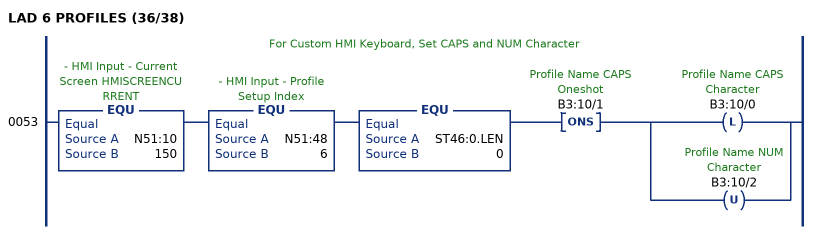
% Rung: 53 %
% For Custom HMI Keyboard, Set CAPS and NUM Character %
SOR EQU N51:10 150 EQU N51:48 6 EQU ST46:0.LEN 0 ONS B3:10/1 BST OTL B3:10/0 NXB OTU B3:10/2 BND EOR
%   N51:10  HMISCREENCURRENT  "- HMI Input - Current Screen" %
%   N51:48  "- HMI Input - Profile Setup Index" %
%   B3:10/1  "Profile Name CAPS Oneshot" %
%   B3:10/0  "Profile Name CAPS Character" %
%   B3:10/2  "Profile Name NUM Character" %

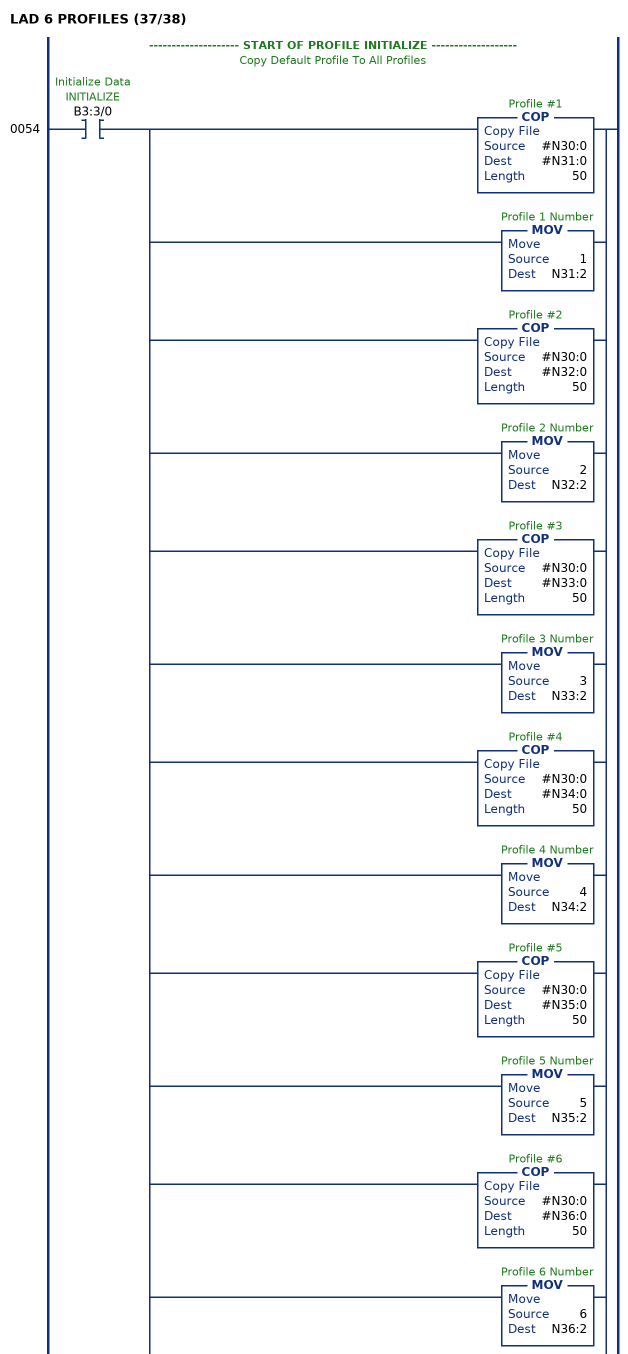

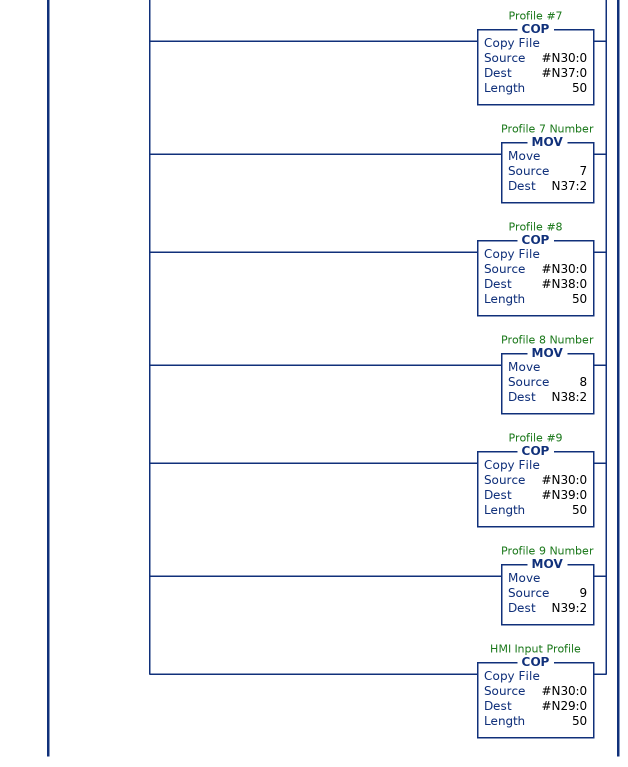
% Rung: 54 %
% TITLE: -------------------- START OF PROFILE INITIALIZE ------------------- %
% Copy Default Profile To All Profiles %
SOR XIC B3:3/0 BST COP #N30:0 #N31:0 50 NXB MOV 1 N31:2 NXB COP #N30:0 #N32:0 50 NXB MOV 2 N32:2 NXB COP #N30:0 #N33:0 50 NXB MOV 3 N33:2 NXB COP #N30:0 #N34:0 50 NXB MOV 4 N34:2 NXB COP #N30:0 #N35:0 50 NXB MOV 5 N35:2 NXB COP #N30:0 #N36:0 50 NXB MOV 6 N36:2 NXB COP #N30:0 #N37:0 50 NXB MOV 7 N37:2 NXB COP #N30:0 #N38:0 50 NXB MOV 8 N38:2 NXB COP #N30:0 #N39:0 50 NXB MOV 9 N39:2 NXB COP #N30:0 #N29:0 50 BND EOR
%   B3:3/0  INITIALIZE  "Initialize Data" %
%   N30:0  "Enable bits" %
%   N31:0  "Profile #1" %
%   N31:2  "Profile 1 Number" %
%   N32:0  "Profile #2" %
%   N32:2  "Profile 2 Number" %
%   N33:0  "Profile #3" %
%   N33:2  "Profile 3 Number" %
%   N34:0  "Profile #4" %
%   N34:2  "Profile 4 Number" %
%   N35:0  "Profile #5" %
%   N35:2  "Profile 5 Number" %
%   N36:0  "Profile #6" %
%   N36:2  "Profile 6 Number" %
%   N37:0  "Profile #7" %
%   N37:2  "Profile 7 Number" %
%   N38:0  "Profile #8" %
%   N38:2  "Profile 8 Number" %
%   N39:0  "Profile #9" %
%   N39:2  "Profile 9 Number" %
%   N29:0  "HMI Input Profile" %

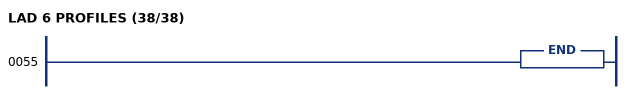
% Rung: 55 %
SOR END EOR

LADDER 7 "OPTIONS"
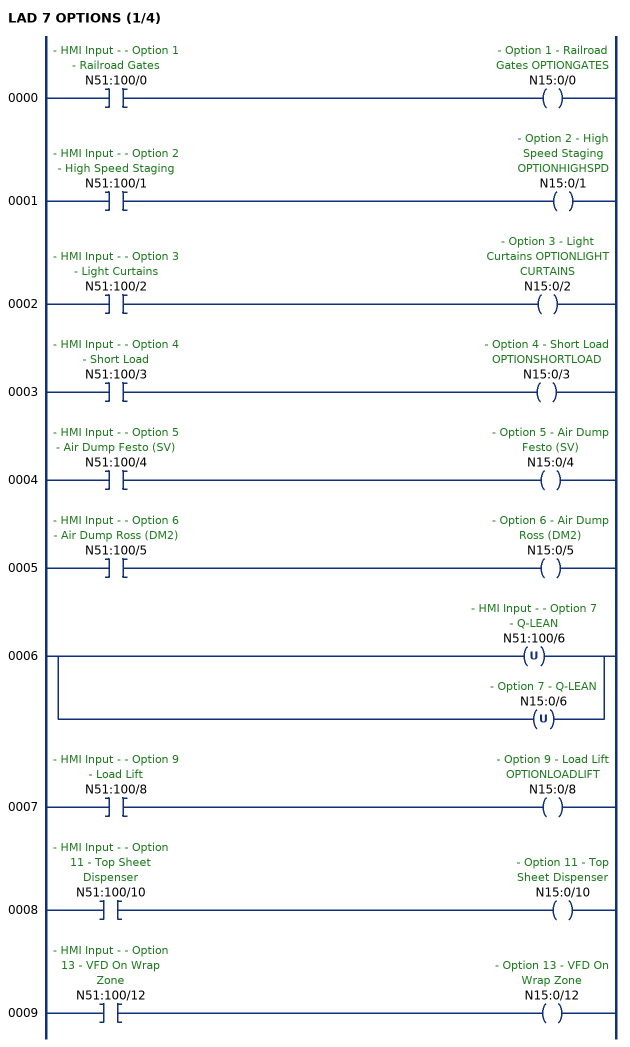
% Rung: 0 %
SOR XIC N51:100/0 OTE N15:0/0 EOR
%   N51:100/0  "- HMI Input - - Option 1 - Railroad Gates" %
%   N15:0/0  OPTIONGATES  "- Option 1 - Railroad Gates" %
% Rung: 1 %
SOR XIC N51:100/1 OTE N15:0/1 EOR
%   N51:100/1  "- HMI Input - - Option 2 - High Speed Staging" %
%   N15:0/1  OPTIONHIGHSPD  "- Option 2 - High Speed Staging" %
% Rung: 2 %
SOR XIC N51:100/2 OTE N15:0/2 EOR
%   N51:100/2  "- HMI Input - - Option 3 - Light Curtains" %
%   N15:0/2  OPTIONLIGHTCURTAINS  "- Option 3 - Light Curtains" %
% Rung: 3 %
SOR XIC N51:100/3 OTE N15:0/3 EOR
%   N51:100/3  "- HMI Input - - Option 4 - Short Load" %
%   N15:0/3  OPTIONSHORTLOAD  "- Option 4 - Short Load" %
% Rung: 4 %
SOR XIC N51:100/4 OTE N15:0/4 EOR
%   N51:100/4  "- HMI Input - - Option 5 - Air Dump Festo (SV)" %
%   N15:0/4  "- Option 5 - Air Dump Festo (SV)" %
% Rung: 5 %
SOR XIC N51:100/5 OTE N15:0/5 EOR
%   N51:100/5  "- HMI Input - - Option 6 - Air Dump Ross (DM2)" %
%   N15:0/5  "- Option 6 - Air Dump Ross (DM2)" %
% Rung: 6 %
SOR BST OTU N51:100/6 NXB OTU N15:0/6 BND EOR
%   N51:100/6  "- HMI Input - - Option 7 - Q-LEAN" %
%   N15:0/6  "- Option 7 - Q-LEAN" %
% Rung: 7 %
SOR XIC N51:100/8 OTE N15:0/8 EOR
%   N51:100/8  "- HMI Input - - Option 9 - Load Lift" %
%   N15:0/8  OPTIONLOADLIFT  "- Option 9 - Load Lift" %
% Rung: 8 %
SOR XIC N51:100/10 OTE N15:0/10 EOR
%   N51:100/10  "- HMI Input - - Option 11 - Top Sheet Dispenser" %
%   N15:0/10  "- Option 11 - Top Sheet Dispenser" %
% Rung: 9 %
SOR XIC N51:100/12 OTE N15:0/12 EOR
%   N51:100/12  "- HMI Input - - Option 13 - VFD On Wrap Zone" %
%   N15:0/12  "- Option 13 - VFD On Wrap Zone" %

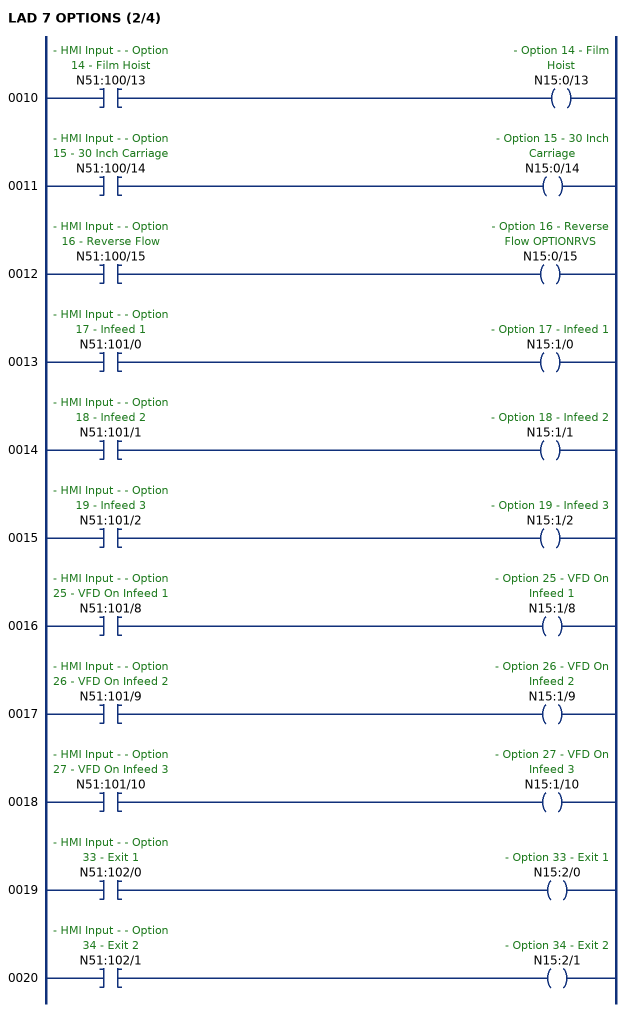
% Rung: 10 %
SOR XIC N51:100/13 OTE N15:0/13 EOR
%   N51:100/13  "- HMI Input - - Option 14 - Film Hoist" %
%   N15:0/13  "- Option 14 - Film Hoist" %
% Rung: 11 %
SOR XIC N51:100/14 OTE N15:0/14 EOR
%   N51:100/14  "- HMI Input - - Option 15 - 30 Inch Carriage" %
%   N15:0/14  "- Option 15 - 30 Inch Carriage" %
% Rung: 12 %
SOR XIC N51:100/15 OTE N15:0/15 EOR
%   N51:100/15  "- HMI Input - - Option 16 - Reverse Flow" %
%   N15:0/15  OPTIONRVS  "- Option 16 - Reverse Flow" %
% Rung: 13 %
SOR XIC N51:101/0 OTE N15:1/0 EOR
%   N51:101/0  "- HMI Input - - Option 17 - Infeed 1" %
%   N15:1/0  "- Option 17 - Infeed 1" %
% Rung: 14 %
SOR XIC N51:101/1 OTE N15:1/1 EOR
%   N51:101/1  "- HMI Input - - Option 18 - Infeed 2" %
%   N15:1/1  "- Option 18 - Infeed 2" %
% Rung: 15 %
SOR XIC N51:101/2 OTE N15:1/2 EOR
%   N51:101/2  "- HMI Input - - Option 19 - Infeed 3" %
%   N15:1/2  "- Option 19 - Infeed 3" %
% Rung: 16 %
SOR XIC N51:101/8 OTE N15:1/8 EOR
%   N51:101/8  "- HMI Input - - Option 25 - VFD On Infeed 1" %
%   N15:1/8  "- Option 25 - VFD On Infeed 1" %
% Rung: 17 %
SOR XIC N51:101/9 OTE N15:1/9 EOR
%   N51:101/9  "- HMI Input - - Option 26 - VFD On Infeed 2" %
%   N15:1/9  "- Option 26 - VFD On Infeed 2" %
% Rung: 18 %
SOR XIC N51:101/10 OTE N15:1/10 EOR
%   N51:101/10  "- HMI Input - - Option 27 - VFD On Infeed 3" %
%   N15:1/10  "- Option 27 - VFD On Infeed 3" %
% Rung: 19 %
SOR XIC N51:102/0 OTE N15:2/0 EOR
%   N51:102/0  "- HMI Input - - Option 33 - Exit 1" %
%   N15:2/0  "- Option 33 - Exit 1" %
% Rung: 20 %
SOR XIC N51:102/1 OTE N15:2/1 EOR
%   N51:102/1  "- HMI Input - - Option 34 - Exit 2" %
%   N15:2/1  "- Option 34 - Exit 2" %

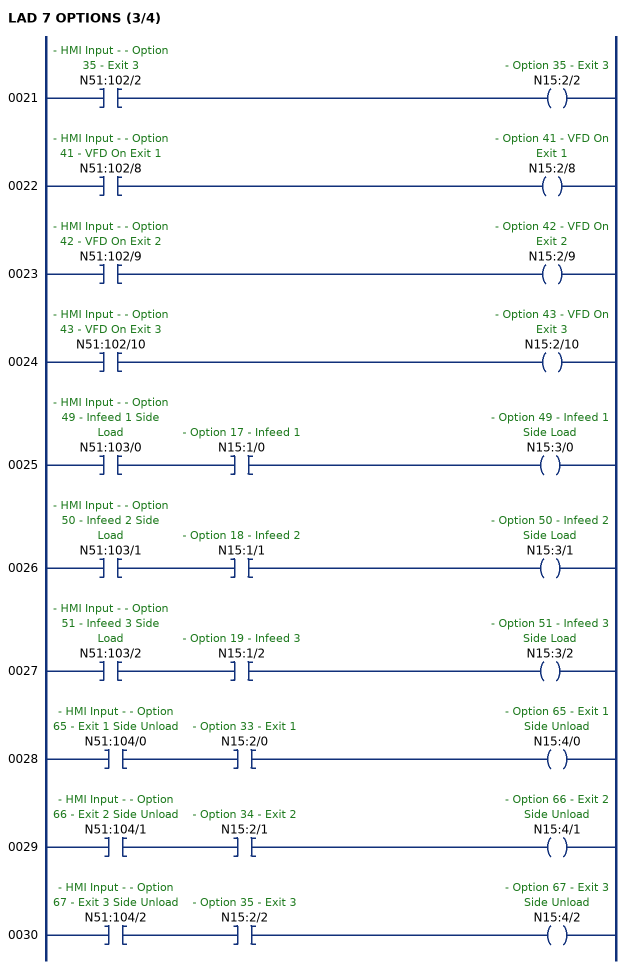
% Rung: 21 %
SOR XIC N51:102/2 OTE N15:2/2 EOR
%   N51:102/2  "- HMI Input - - Option 35 - Exit 3" %
%   N15:2/2  "- Option 35 - Exit 3" %
% Rung: 22 %
SOR XIC N51:102/8 OTE N15:2/8 EOR
%   N51:102/8  "- HMI Input - - Option 41 - VFD On Exit 1" %
%   N15:2/8  "- Option 41 - VFD On Exit 1" %
% Rung: 23 %
SOR XIC N51:102/9 OTE N15:2/9 EOR
%   N51:102/9  "- HMI Input - - Option 42 - VFD On Exit 2" %
%   N15:2/9  "- Option 42 - VFD On Exit 2" %
% Rung: 24 %
SOR XIC N51:102/10 OTE N15:2/10 EOR
%   N51:102/10  "- HMI Input - - Option 43 - VFD On Exit 3" %
%   N15:2/10  "- Option 43 - VFD On Exit 3" %
% Rung: 25 %
SOR XIC N51:103/0 XIC N15:1/0 OTE N15:3/0 EOR
%   N51:103/0  "- HMI Input - - Option 49 - Infeed 1 Side Load" %
%   N15:1/0  "- Option 17 - Infeed 1" %
%   N15:3/0  "- Option 49 - Infeed 1 Side Load" %
% Rung: 26 %
SOR XIC N51:103/1 XIC N15:1/1 OTE N15:3/1 EOR
%   N51:103/1  "- HMI Input - - Option 50 - Infeed 2 Side Load" %
%   N15:1/1  "- Option 18 - Infeed 2" %
%   N15:3/1  "- Option 50 - Infeed 2 Side Load" %
% Rung: 27 %
SOR XIC N51:103/2 XIC N15:1/2 OTE N15:3/2 EOR
%   N51:103/2  "- HMI Input - - Option 51 - Infeed 3 Side Load" %
%   N15:1/2  "- Option 19 - Infeed 3" %
%   N15:3/2  "- Option 51 - Infeed 3 Side Load" %
% Rung: 28 %
SOR XIC N51:104/0 XIC N15:2/0 OTE N15:4/0 EOR
%   N51:104/0  "- HMI Input - - Option 65 - Exit 1 Side Unload" %
%   N15:2/0  "- Option 33 - Exit 1" %
%   N15:4/0  "- Option 65 - Exit 1 Side Unload" %
% Rung: 29 %
SOR XIC N51:104/1 XIC N15:2/1 OTE N15:4/1 EOR
%   N51:104/1  "- HMI Input - - Option 66 - Exit 2 Side Unload" %
%   N15:2/1  "- Option 34 - Exit 2" %
%   N15:4/1  "- Option 66 - Exit 2 Side Unload" %
% Rung: 30 %
SOR XIC N51:104/2 XIC N15:2/2 OTE N15:4/2 EOR
%   N51:104/2  "- HMI Input - - Option 67 - Exit 3 Side Unload" %
%   N15:2/2  "- Option 35 - Exit 3" %
%   N15:4/2  "- Option 67 - Exit 3 Side Unload" %

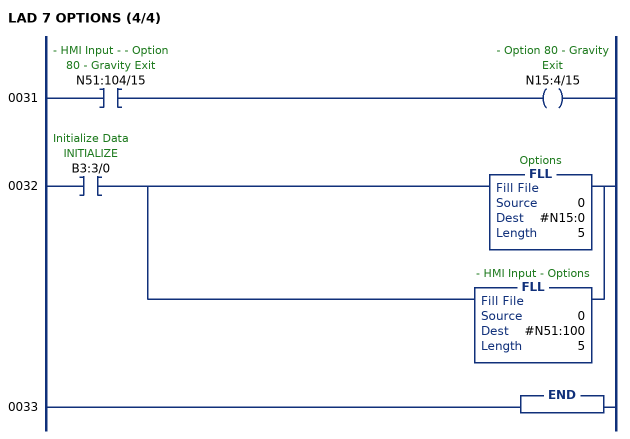
% Rung: 31 %
SOR XIC N51:104/15 OTE N15:4/15 EOR
%   N51:104/15  "- HMI Input - - Option 80 - Gravity Exit" %
%   N15:4/15  "- Option 80 - Gravity Exit" %
% Rung: 32 %
SOR XIC B3:3/0 BST FLL 0 #N15:0 5 NXB FLL 0 #N51:100 5 BND EOR
%   B3:3/0  INITIALIZE  "Initialize Data" %
%   N15:0  "Options" %
%   N51:100  "- HMI Input - Options" %
% Rung: 33 %
SOR END EOR

LADDER 8 "CONSTANTS"
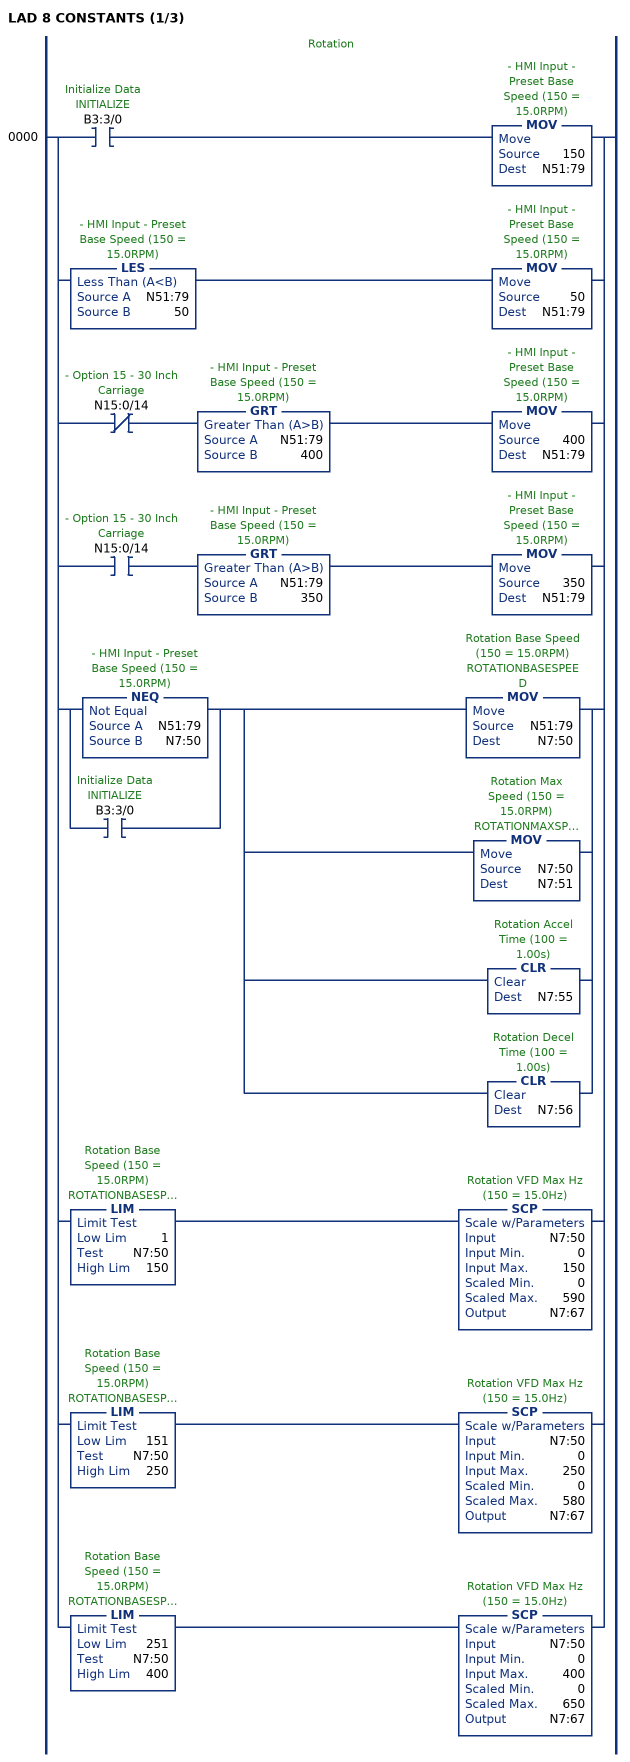
% Rung: 0 %
% Rotation %
SOR BST BST XIC B3:3/0 MOV 150 N51:79 NXB LES N51:79 50 MOV 50 N51:79 NXB XIO N15:0/14 GRT N51:79 400 MOV 400 N51:79 NXB XIC N15:0/14 GRT N51:79 350 MOV 350 N51:79 BND NXB BST NEQ N51:79 N7:50 NXB XIC B3:3/0 BND BST MOV N51:79 N7:50 NXB MOV N7:50 N7:51 NXB CLR N7:55 NXB CLR N7:56 BND NXB BST LIM 1 N7:50 150 SCP N7:50 0 150 0 590 N7:67 NXB LIM 151 N7:50 250 SCP N7:50 0 250 0 580 N7:67 NXB LIM 251 N7:50 400 SCP N7:50 0 400 0 650 N7:67 BND BND EOR
%   B3:3/0  INITIALIZE  "Initialize Data" %
%   N51:79  "- HMI Input - Preset Base Speed (150 = 15.0RPM)" %
%   N15:0/14  "- Option 15 - 30 Inch Carriage" %
%   N7:50  ROTATIONBASESPEED  "Rotation Base Speed (150 = 15.0RPM)" %
%   N7:51  ROTATIONMAXSPEED  "Rotation Max Speed (150 = 15.0RPM)" %
%   N7:55  "Rotation Accel Time (100 = 1.00s)" %
%   N7:56  "Rotation Decel Time (100 = 1.00s)" %
%   N7:67  "Rotation VFD Max Hz (150 = 15.0Hz)" %

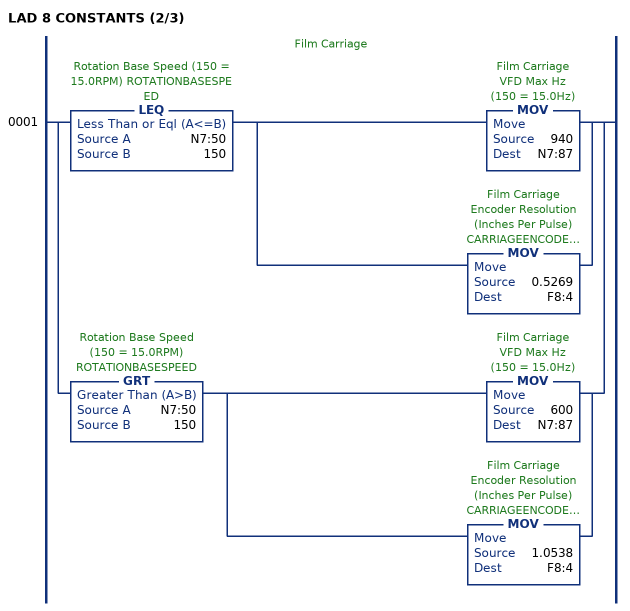
% Rung: 1 %
% Film Carriage %
SOR BST LEQ N7:50 150 BST MOV 940 N7:87 NXB MOV 0.5269 F8:4 BND NXB GRT N7:50 150 BST MOV 600 N7:87 NXB MOV 1.0538 F8:4 BND BND EOR
%   N7:50  ROTATIONBASESPEED  "Rotation Base Speed (150 = 15.0RPM)" %
%   N7:87  "Film Carriage VFD Max Hz (150 = 15.0Hz)" %
%   F8:4  CARRIAGEENCODERRES  "Film Carriage Encoder Resolution (Inches Per Pulse)" %

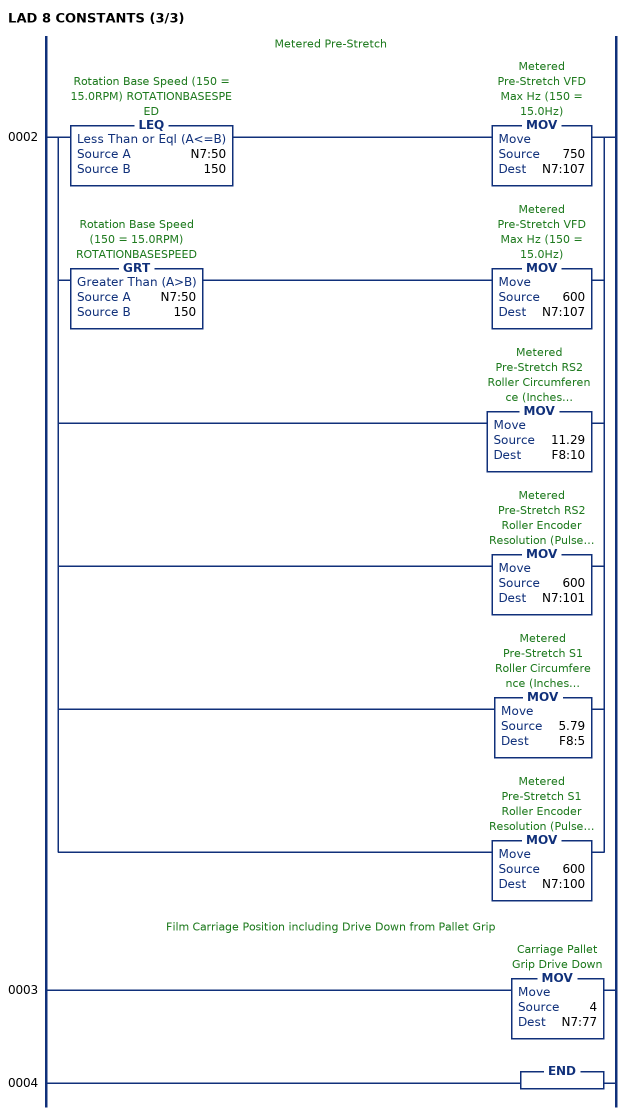
% Rung: 2 %
% Metered Pre-Stretch %
SOR BST BST LEQ N7:50 150 MOV 750 N7:107 NXB GRT N7:50 150 MOV 600 N7:107 BND NXB MOV 11.29 F8:10 NXB MOV 600 N7:101 NXB MOV 5.79 F8:5 NXB MOV 600 N7:100 BND EOR
%   N7:50  ROTATIONBASESPEED  "Rotation Base Speed (150 = 15.0RPM)" %
%   N7:107  "Metered Pre-Stretch VFD Max Hz (150 = 15.0Hz)" %
%   F8:10  MPSRS2CIRC  "Metered Pre-Stretch RS2 Roller Circumference (Inches)" %
%   N7:101  MPSRS2ENCODERRES  "Metered Pre-Stretch RS2 Roller Encoder Resolution (Pulses Per Rev)" %
%   F8:5  MPSS1CIRC  "Metered Pre-Stretch S1 Roller Circumference (Inches)" %
%   N7:100  MPSS1ENCODERRES  "Metered Pre-Stretch S1 Roller Encoder Resolution (Pulses Per Rev)" %
% Rung: 3 %
% Film Carriage Position including Drive Down from Pallet Grip %
SOR MOV 4 N7:77 EOR
%   N7:77  "Carriage Pallet Grip Drive Down" %
% Rung: 4 %
SOR END EOR

LADDER 9 "WRAP CYCLE"
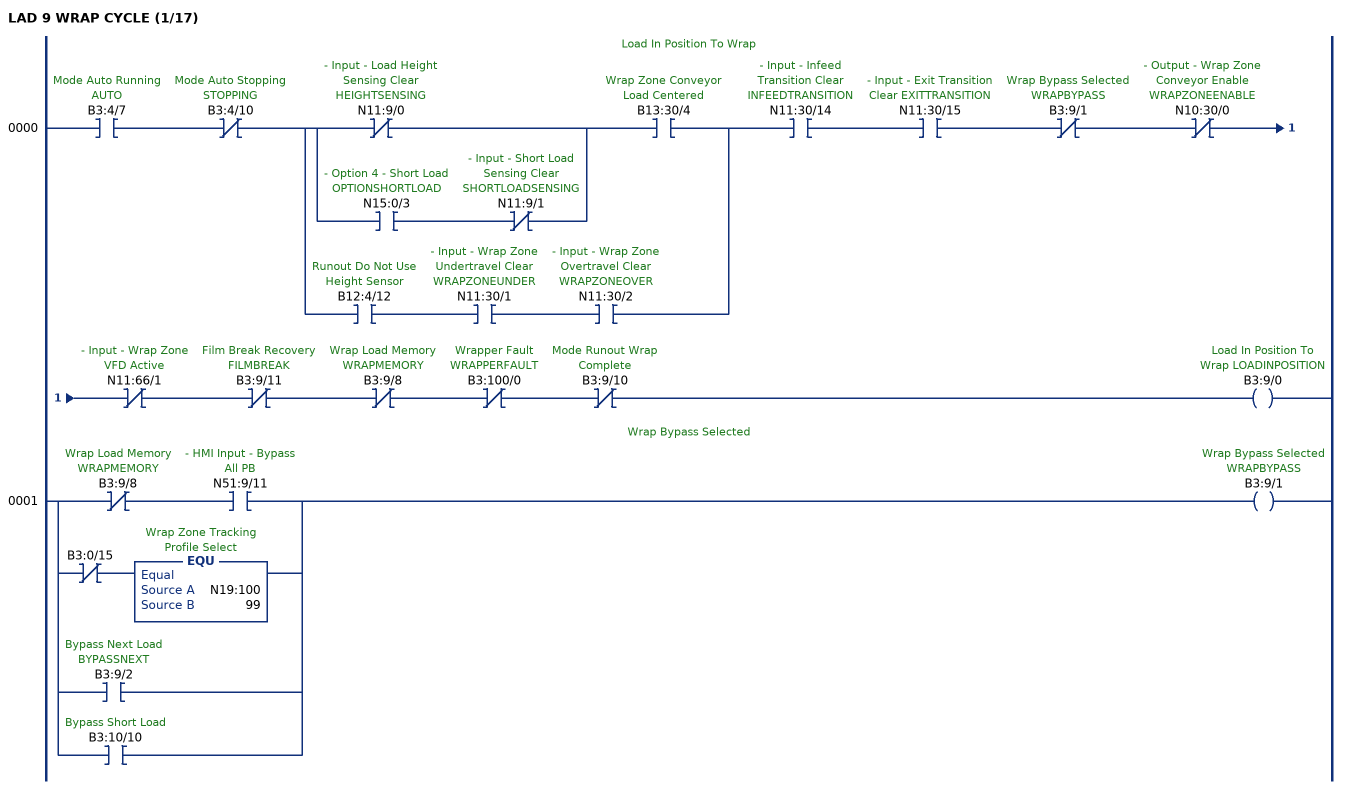
% Rung: 0 %
% Load In Position To Wrap %
SOR XIC B3:4/7 XIO B3:4/10 BST BST XIO N11:9/0 NXB XIC N15:0/3 XIO N11:9/1 BND XIC B13:30/4 NXB XIC B12:4/12 XIC N11:30/1 XIC N11:30/2 BND XIC N11:30/14 XIC N11:30/15 XIO B3:9/1 XIO N10:30/0 XIO N11:66/1 XIO B3:9/11 XIO B3:9/8 XIO B3:100/0 XIO B3:9/10 OTE B3:9/0 EOR
%   B3:4/7  AUTO  "Mode Auto Running" %
%   B3:4/10  STOPPING  "Mode Auto Stopping" %
%   N11:9/0  HEIGHTSENSING  "- Input - Load Height Sensing Clear" %
%   N15:0/3  OPTIONSHORTLOAD  "- Option 4 - Short Load" %
%   N11:9/1  SHORTLOADSENSING  "- Input - Short Load Sensing Clear" %
%   B13:30/4  "Wrap Zone Conveyor Load Centered" %
%   B12:4/12  "Runout Do Not Use Height Sensor" %
%   N11:30/1  WRAPZONEUNDER  "- Input - Wrap Zone Undertravel Clear" %
%   N11:30/2  WRAPZONEOVER  "- Input - Wrap Zone Overtravel Clear" %
%   N11:30/14  INFEEDTRANSITION  "- Input - Infeed Transition Clear" %
%   N11:30/15  EXITTRANSITION  "- Input - Exit Transition Clear" %
%   B3:9/1  WRAPBYPASS  "Wrap Bypass Selected" %
%   N10:30/0  WRAPZONEENABLE  "- Output - Wrap Zone Conveyor Enable" %
%   N11:66/1  "- Input - Wrap Zone VFD Active" %
%   B3:9/11  FILMBREAK  "Film Break Recovery" %
%   B3:9/8  WRAPMEMORY  "Wrap Load Memory" %
%   B3:100/0  WRAPPERFAULT  "Wrapper Fault" %
%   B3:9/10  "Mode Runout Wrap Complete" %
%   B3:9/0  LOADINPOSITION  "Load In Position To Wrap" %
% Rung: 1 %
% Wrap Bypass Selected %
SOR BST XIO B3:9/8 XIC N51:9/11 NXB XIO B3:0/15 EQU N19:100 99 NXB XIC B3:9/2 NXB XIC B3:10/10 BND OTE B3:9/1 EOR
%   B3:9/8  WRAPMEMORY  "Wrap Load Memory" %
%   N51:9/11  "- HMI Input - Bypass All PB" %
%   N19:100  "Wrap Zone Tracking Profile Select" %
%   B3:9/2  BYPASSNEXT  "Bypass Next Load" %
%   B3:10/10  "Bypass Short Load" %
%   B3:9/1  WRAPBYPASS  "Wrap Bypass Selected" %

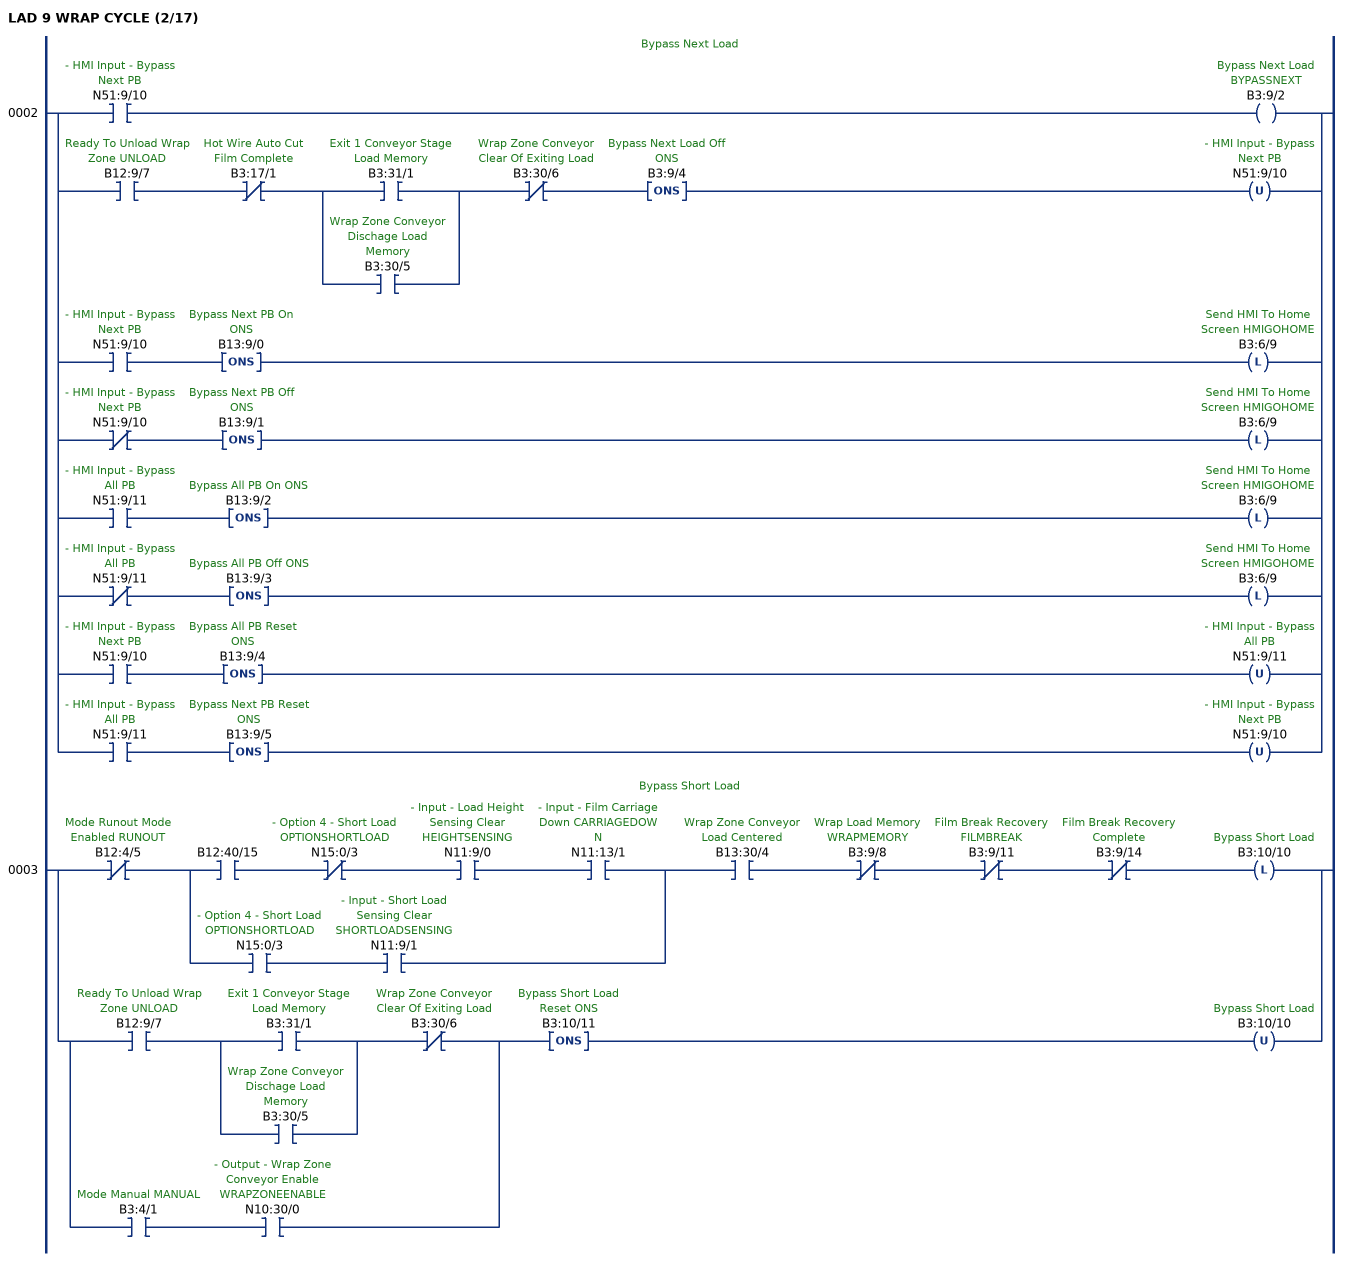
% Rung: 2 %
% Bypass Next Load %
SOR BST XIC N51:9/10 OTE B3:9/2 NXB XIC B12:9/7 XIO B3:17/1 BST XIC B3:31/1 NXB XIC B3:30/5 BND XIO B3:30/6 ONS B3:9/4 OTU N51:9/10 NXB BST XIC N51:9/10 ONS B13:9/0 OTL B3:6/9 NXB XIO N51:9/10 ONS B13:9/1 OTL B3:6/9 NXB XIC N51:9/11 ONS B13:9/2 OTL B3:6/9 NXB XIO N51:9/11 ONS B13:9/3 OTL B3:6/9 BND NXB BST XIC N51:9/10 ONS B13:9/4 OTU N51:9/11 NXB XIC N51:9/11 ONS B13:9/5 OTU N51:9/10 BND BND EOR
%   N51:9/10  "- HMI Input - Bypass Next PB" %
%   B3:9/2  BYPASSNEXT  "Bypass Next Load" %
%   B12:9/7  UNLOAD  "Ready To Unload Wrap Zone" %
%   B3:17/1  "Hot Wire Auto Cut Film Complete" %
%   B3:31/1  "Exit 1 Conveyor Stage Load Memory" %
%   B3:30/5  "Wrap Zone Conveyor Dischage Load Memory" %
%   B3:30/6  "Wrap Zone Conveyor Clear Of Exiting Load" %
%   B3:9/4  "Bypass Next Load Off ONS" %
%   B13:9/0  "Bypass Next PB On ONS" %
%   B3:6/9  HMIGOHOME  "Send HMI To Home Screen" %
%   B13:9/1  "Bypass Next PB Off ONS" %
%   N51:9/11  "- HMI Input - Bypass All PB" %
%   B13:9/2  "Bypass All PB On ONS" %
%   B13:9/3  "Bypass All PB Off ONS" %
%   B13:9/4  "Bypass All PB Reset ONS" %
%   B13:9/5  "Bypass Next PB Reset ONS" %
% Rung: 3 %
% Bypass Short Load %
SOR BST XIO B12:4/5 BST XIC B12:40/15 XIO N15:0/3 XIC N11:9/0 XIC N11:13/1 NXB XIC N15:0/3 XIC N11:9/1 BND XIC B13:30/4 XIO B3:9/8 XIO B3:9/11 XIO B3:9/14 OTL B3:10/10 NXB BST XIC B12:9/7 BST XIC B3:31/1 NXB XIC B3:30/5 BND XIO B3:30/6 NXB XIC B3:4/1 XIC N10:30/0 BND ONS B3:10/11 OTU B3:10/10 BND EOR
%   B12:4/5  RUNOUT  "Mode Runout Mode Enabled" %
%   N15:0/3  OPTIONSHORTLOAD  "- Option 4 - Short Load" %
%   N11:9/0  HEIGHTSENSING  "- Input - Load Height Sensing Clear" %
%   N11:13/1  CARRIAGEDOWN  "- Input - Film Carriage Down" %
%   N11:9/1  SHORTLOADSENSING  "- Input - Short Load Sensing Clear" %
%   B13:30/4  "Wrap Zone Conveyor Load Centered" %
%   B3:9/8  WRAPMEMORY  "Wrap Load Memory" %
%   B3:9/11  FILMBREAK  "Film Break Recovery" %
%   B3:9/14  "Film Break Recovery Complete" %
%   B3:10/10  "Bypass Short Load" %
%   B12:9/7  UNLOAD  "Ready To Unload Wrap Zone" %
%   B3:31/1  "Exit 1 Conveyor Stage Load Memory" %
%   B3:30/5  "Wrap Zone Conveyor Dischage Load Memory" %
%   B3:30/6  "Wrap Zone Conveyor Clear Of Exiting Load" %
%   B3:4/1  MANUAL  "Mode Manual" %
%   N10:30/0  WRAPZONEENABLE  "- Output - Wrap Zone Conveyor Enable" %
%   B3:10/11  "Bypass Short Load Reset ONS" %

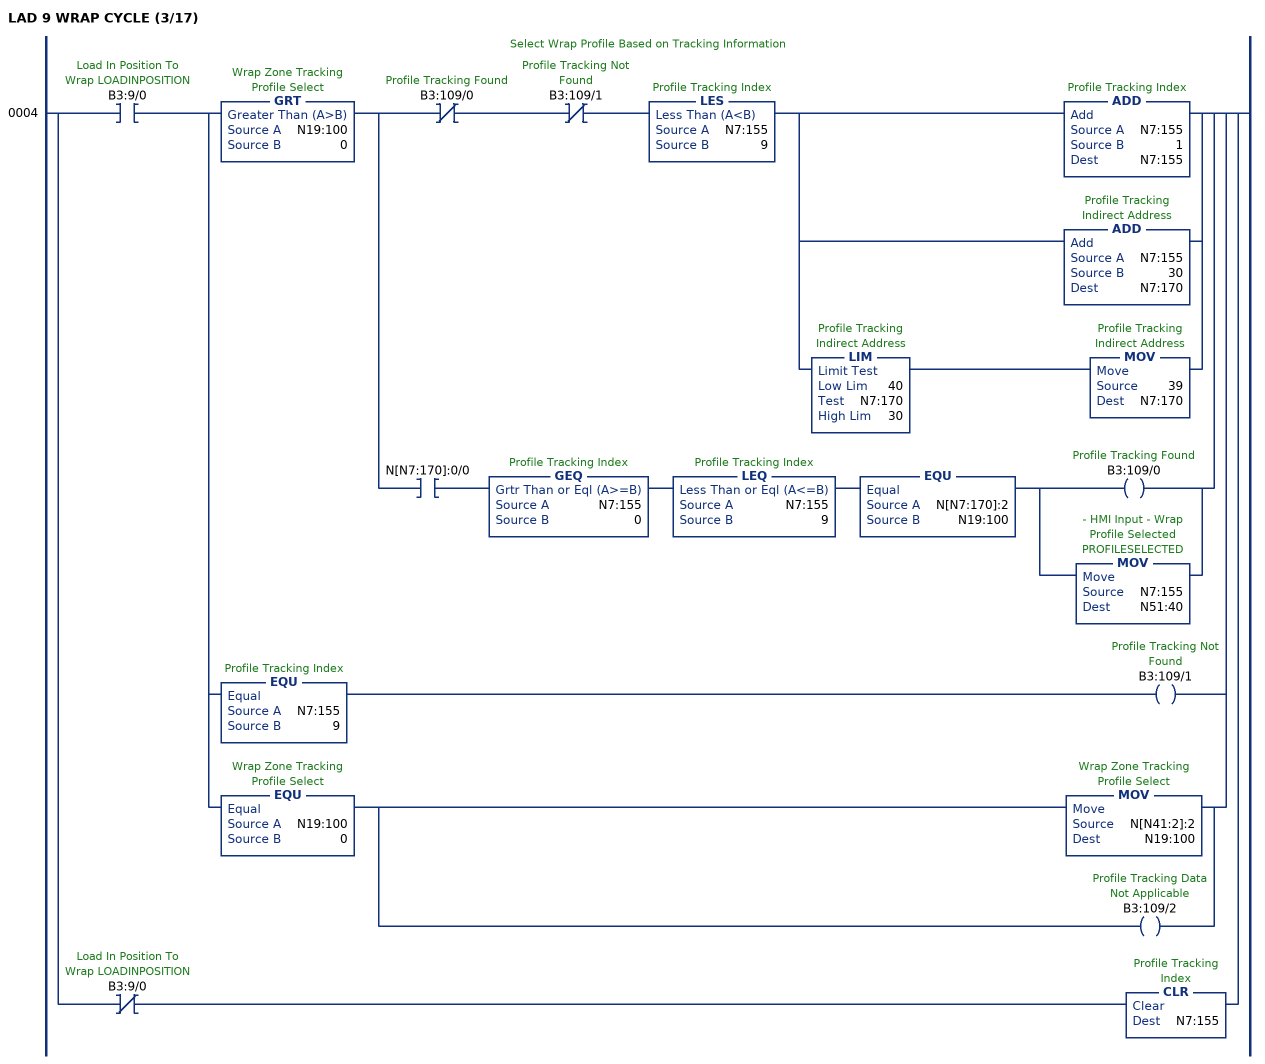
% Rung: 4 %
% Select Wrap Profile Based on Tracking Information %
SOR BST XIC B3:9/0 BST GRT N19:100 0 BST XIO B3:109/0 XIO B3:109/1 LES N7:155 9 BST ADD N7:155 1 N7:155 NXB ADD N7:155 30 N7:170 NXB LIM 40 N7:170 30 MOV 39 N7:170 BND NXB XIC N[N7:170]:0/0 GEQ N7:155 0 LEQ N7:155 9 EQU N[N7:170]:2 N19:100 BST OTE B3:109/0 NXB MOV N7:155 N51:40 BND BND NXB EQU N7:155 9 OTE B3:109/1 NXB EQU N19:100 0 BST MOV N[N41:2]:2 N19:100 NXB OTE B3:109/2 BND BND NXB XIO B3:9/0 CLR N7:155 BND EOR
%   B3:9/0  LOADINPOSITION  "Load In Position To Wrap" %
%   N19:100  "Wrap Zone Tracking Profile Select" %
%   B3:109/0  "Profile Tracking Found" %
%   B3:109/1  "Profile Tracking Not Found" %
%   N7:155  "Profile Tracking Index" %
%   N7:170  "Profile Tracking Indirect Address" %
%   N51:40  PROFILESELECTED  "- HMI Input - Wrap Profile Selected" %
%   N41:2  "Profile Selected Indirect Address" %
%   B3:109/2  "Profile Tracking Data Not Applicable" %

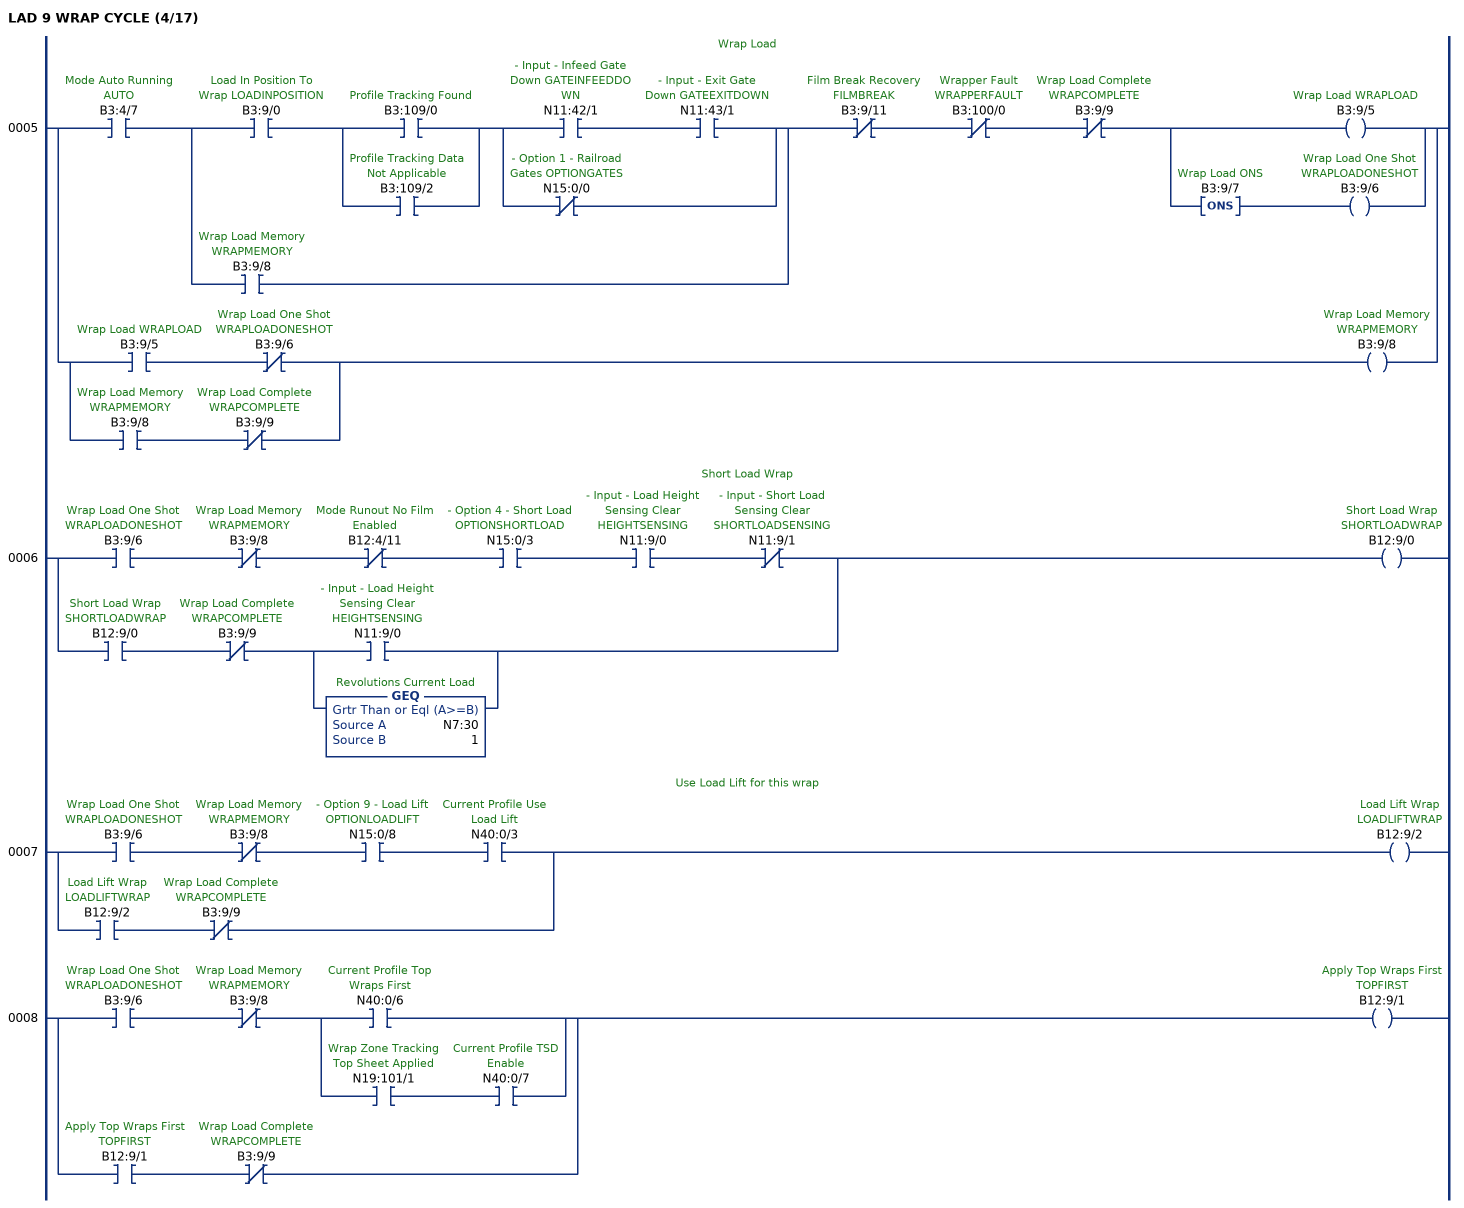
% Rung: 5 %
% Wrap Load %
SOR BST XIC B3:4/7 BST XIC B3:9/0 BST XIC B3:109/0 NXB XIC B3:109/2 BND BST XIC N11:42/1 XIC N11:43/1 NXB XIO N15:0/0 BND NXB XIC B3:9/8 BND XIO B3:9/11 XIO B3:100/0 XIO B3:9/9 BST OTE B3:9/5 NXB ONS B3:9/7 OTE B3:9/6 BND NXB BST XIC B3:9/5 XIO B3:9/6 NXB XIC B3:9/8 XIO B3:9/9 BND OTE B3:9/8 BND EOR
%   B3:4/7  AUTO  "Mode Auto Running" %
%   B3:9/0  LOADINPOSITION  "Load In Position To Wrap" %
%   B3:109/0  "Profile Tracking Found" %
%   B3:109/2  "Profile Tracking Data Not Applicable" %
%   N11:42/1  GATEINFEEDDOWN  "- Input - Infeed Gate Down" %
%   N11:43/1  GATEEXITDOWN  "- Input - Exit Gate Down" %
%   N15:0/0  OPTIONGATES  "- Option 1 - Railroad Gates" %
%   B3:9/8  WRAPMEMORY  "Wrap Load Memory" %
%   B3:9/11  FILMBREAK  "Film Break Recovery" %
%   B3:100/0  WRAPPERFAULT  "Wrapper Fault" %
%   B3:9/9  WRAPCOMPLETE  "Wrap Load Complete" %
%   B3:9/5  WRAPLOAD  "Wrap Load" %
%   B3:9/7  "Wrap Load ONS" %
%   B3:9/6  WRAPLOADONESHOT  "Wrap Load One Shot" %
% Rung: 6 %
% Short Load Wrap %
SOR BST XIC B3:9/6 XIO B3:9/8 XIO B12:4/11 XIC N15:0/3 XIC N11:9/0 XIO N11:9/1 NXB XIC B12:9/0 XIO B3:9/9 BST XIC N11:9/0 NXB GEQ N7:30 1 BND BND OTE B12:9/0 EOR
%   B3:9/6  WRAPLOADONESHOT  "Wrap Load One Shot" %
%   B3:9/8  WRAPMEMORY  "Wrap Load Memory" %
%   B12:4/11  "Mode Runout No Film Enabled" %
%   N15:0/3  OPTIONSHORTLOAD  "- Option 4 - Short Load" %
%   N11:9/0  HEIGHTSENSING  "- Input - Load Height Sensing Clear" %
%   N11:9/1  SHORTLOADSENSING  "- Input - Short Load Sensing Clear" %
%   B12:9/0  SHORTLOADWRAP  "Short Load Wrap" %
%   B3:9/9  WRAPCOMPLETE  "Wrap Load Complete" %
%   N7:30  "Revolutions Current Load" %
% Rung: 7 %
% Use Load Lift for this wrap %
SOR BST XIC B3:9/6 XIO B3:9/8 XIC N15:0/8 XIC N40:0/3 NXB XIC B12:9/2 XIO B3:9/9 BND OTE B12:9/2 EOR
%   B3:9/6  WRAPLOADONESHOT  "Wrap Load One Shot" %
%   B3:9/8  WRAPMEMORY  "Wrap Load Memory" %
%   N15:0/8  OPTIONLOADLIFT  "- Option 9 - Load Lift" %
%   N40:0/3  "Current Profile Use Load Lift" %
%   B12:9/2  LOADLIFTWRAP  "Load Lift Wrap" %
%   B3:9/9  WRAPCOMPLETE  "Wrap Load Complete" %
% Rung: 8 %
SOR BST XIC B3:9/6 XIO B3:9/8 BST XIC N40:0/6 NXB XIC N19:101/1 XIC N40:0/7 BND NXB XIC B12:9/1 XIO B3:9/9 BND OTE B12:9/1 EOR
%   B3:9/6  WRAPLOADONESHOT  "Wrap Load One Shot" %
%   B3:9/8  WRAPMEMORY  "Wrap Load Memory" %
%   N40:0/6  "Current Profile Top Wraps First" %
%   N19:101/1  "Wrap Zone Tracking Top Sheet Applied" %
%   N40:0/7  "Current Profile TSD Enable" %
%   B12:9/1  TOPFIRST  "Apply Top Wraps First" %
%   B3:9/9  WRAPCOMPLETE  "Wrap Load Complete" %

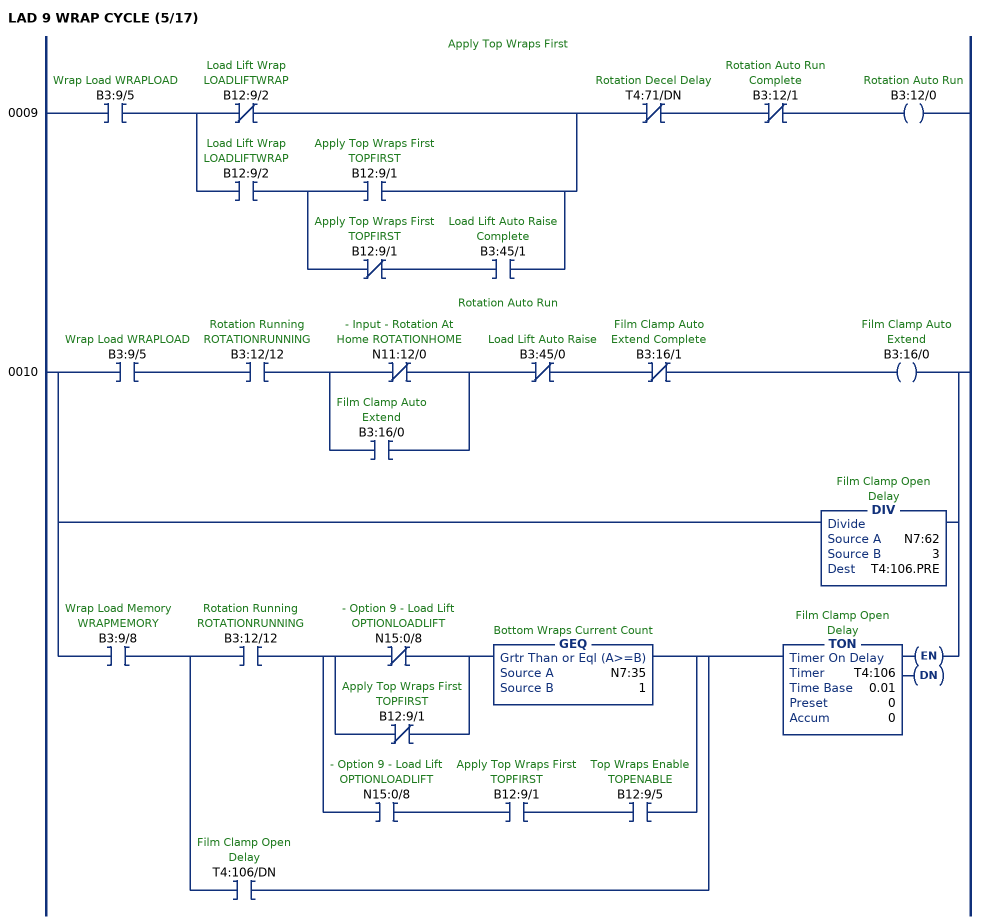
% Rung: 9 %
% Apply Top Wraps First %
SOR XIC B3:9/5 BST XIO B12:9/2 NXB XIC B12:9/2 BST XIC B12:9/1 NXB XIO B12:9/1 XIC B3:45/1 BND BND XIO T4:71/DN XIO B3:12/1 OTE B3:12/0 EOR
%   B3:9/5  WRAPLOAD  "Wrap Load" %
%   B12:9/2  LOADLIFTWRAP  "Load Lift Wrap" %
%   B12:9/1  TOPFIRST  "Apply Top Wraps First" %
%   B3:45/1  "Load Lift Auto Raise Complete" %
%   T4:71  "Rotation Decel Delay" %
%   B3:12/1  "Rotation Auto Run Complete" %
%   B3:12/0  "Rotation Auto Run" %
% Rung: 10 %
% Rotation Auto Run %
SOR BST XIC B3:9/5 XIC B3:12/12 BST XIO N11:12/0 NXB XIC B3:16/0 BND XIO B3:45/0 XIO B3:16/1 OTE B3:16/0 NXB DIV N7:62 3 T4:106.PRE NXB XIC B3:9/8 BST XIC B3:12/12 BST BST XIO N15:0/8 NXB XIO B12:9/1 BND GEQ N7:35 1 NXB XIC N15:0/8 XIC B12:9/1 XIC B12:9/5 BND NXB XIC T4:106/DN BND TON T4:106 0.01 0 0 BND EOR
%   B3:9/5  WRAPLOAD  "Wrap Load" %
%   B3:12/12  ROTATIONRUNNING  "Rotation Running" %
%   N11:12/0  ROTATIONHOME  "- Input - Rotation At Home" %
%   B3:16/0  "Film Clamp Auto Extend" %
%   B3:45/0  "Load Lift Auto Raise" %
%   B3:16/1  "Film Clamp Auto Extend Complete" %
%   N7:62  "Rotation Revolution Time (100 = 1.00s)" %
%   T4:106  "Film Clamp Open Delay" %
%   B3:9/8  WRAPMEMORY  "Wrap Load Memory" %
%   N15:0/8  OPTIONLOADLIFT  "- Option 9 - Load Lift" %
%   B12:9/1  TOPFIRST  "Apply Top Wraps First" %
%   N7:35  "Bottom Wraps Current Count" %
%   B12:9/5  TOPENABLE  "Top Wraps Enable" %

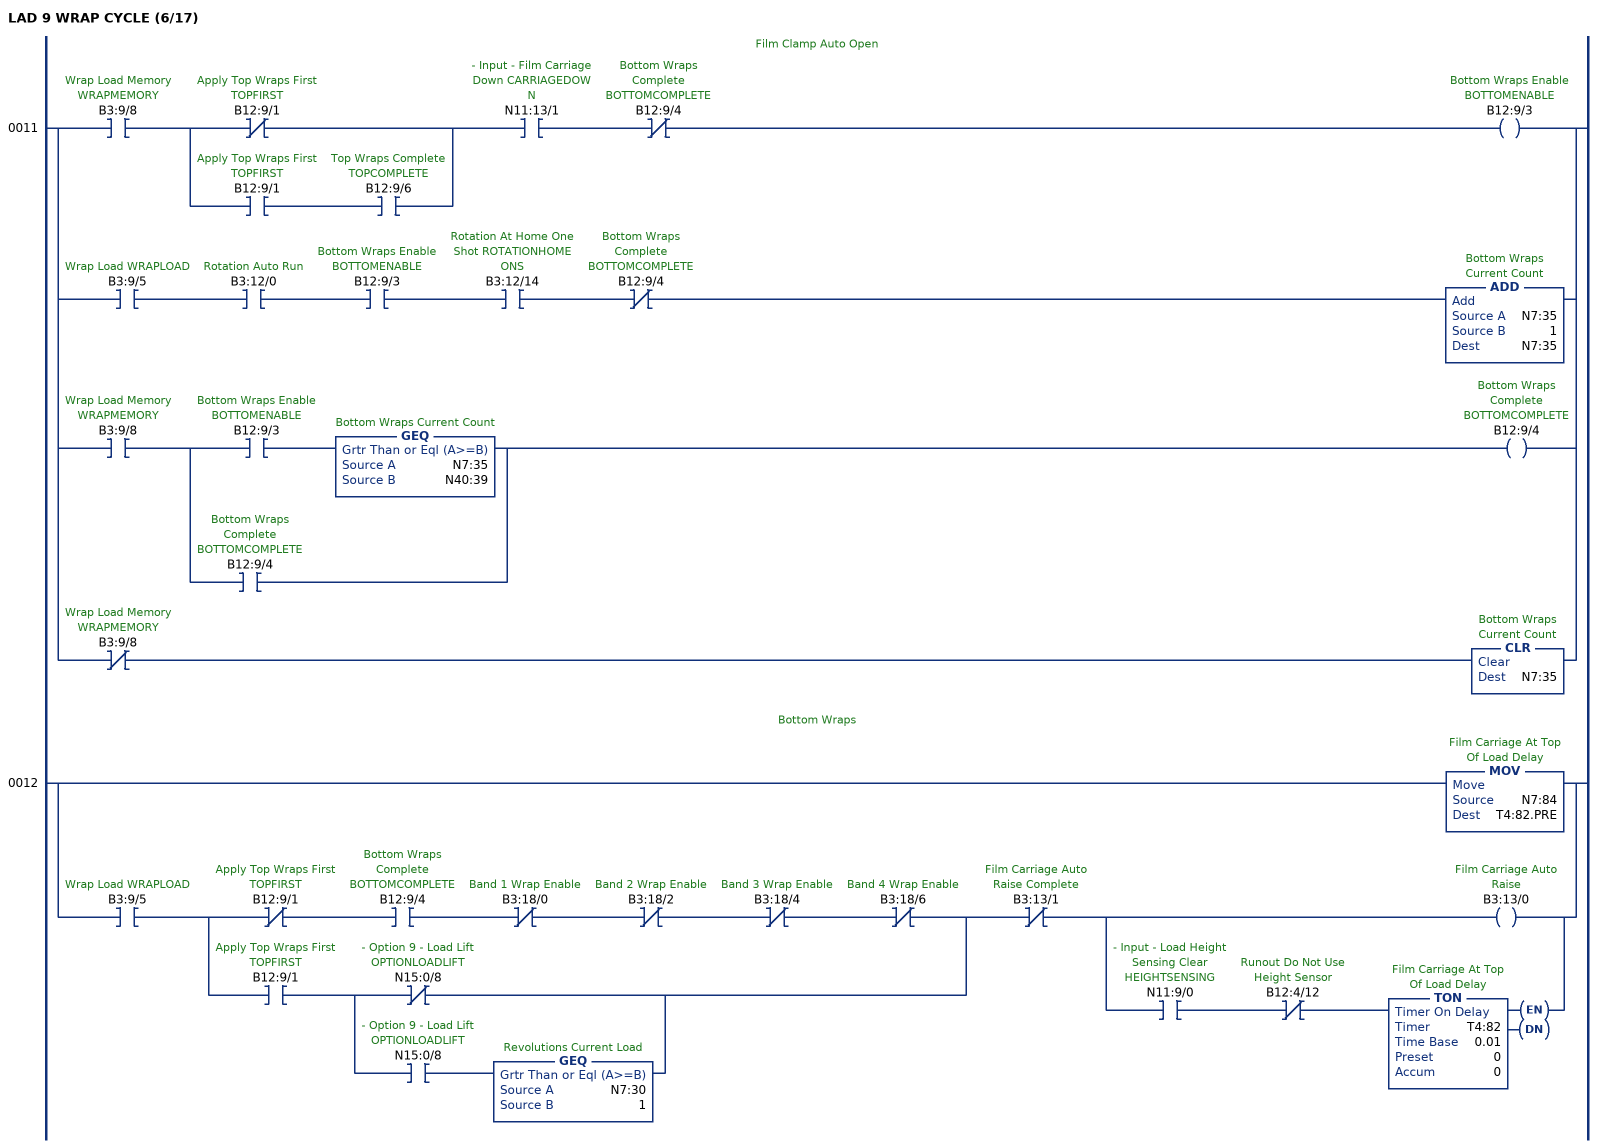
% Rung: 11 %
% Film Clamp Auto Open %
SOR BST XIC B3:9/8 BST XIO B12:9/1 NXB XIC B12:9/1 XIC B12:9/6 BND XIC N11:13/1 XIO B12:9/4 OTE B12:9/3 NXB XIC B3:9/5 XIC B3:12/0 XIC B12:9/3 XIC B3:12/14 XIO B12:9/4 ADD N7:35 1 N7:35 NXB XIC B3:9/8 BST XIC B12:9/3 GEQ N7:35 N40:39 NXB XIC B12:9/4 BND OTE B12:9/4 NXB XIO B3:9/8 CLR N7:35 BND EOR
%   B3:9/8  WRAPMEMORY  "Wrap Load Memory" %
%   B12:9/1  TOPFIRST  "Apply Top Wraps First" %
%   B12:9/6  TOPCOMPLETE  "Top Wraps Complete" %
%   N11:13/1  CARRIAGEDOWN  "- Input - Film Carriage Down" %
%   B12:9/4  BOTTOMCOMPLETE  "Bottom Wraps Complete" %
%   B12:9/3  BOTTOMENABLE  "Bottom Wraps Enable" %
%   B3:9/5  WRAPLOAD  "Wrap Load" %
%   B3:12/0  "Rotation Auto Run" %
%   B3:12/14  ROTATIONHOMEONS  "Rotation At Home One Shot" %
%   N7:35  "Bottom Wraps Current Count" %
% Rung: 12 %
% Bottom Wraps %
SOR BST MOV N7:84 T4:82.PRE NXB XIC B3:9/5 BST XIO B12:9/1 XIC B12:9/4 XIO B3:18/0 XIO B3:18/2 XIO B3:18/4 XIO B3:18/6 NXB XIC B12:9/1 BST XIO N15:0/8 NXB XIC N15:0/8 GEQ N7:30 1 BND BND XIO B3:13/1 BST OTE B3:13/0 NXB XIC N11:9/0 XIO B12:4/12 TON T4:82 0.01 0 0 BND BND EOR
%   N7:84  "Film Carriage Top Of Load Preset (100 = 1.00s)" %
%   T4:82  "Film Carriage At Top Of Load Delay" %
%   B3:9/5  WRAPLOAD  "Wrap Load" %
%   B12:9/1  TOPFIRST  "Apply Top Wraps First" %
%   B12:9/4  BOTTOMCOMPLETE  "Bottom Wraps Complete" %
%   B3:18/0  "Band 1 Wrap Enable" %
%   B3:18/2  "Band 2 Wrap Enable" %
%   B3:18/4  "Band 3 Wrap Enable" %
%   B3:18/6  "Band 4 Wrap Enable" %
%   N15:0/8  OPTIONLOADLIFT  "- Option 9 - Load Lift" %
%   N7:30  "Revolutions Current Load" %
%   B3:13/1  "Film Carriage Auto Raise Complete" %
%   B3:13/0  "Film Carriage Auto Raise" %
%   N11:9/0  HEIGHTSENSING  "- Input - Load Height Sensing Clear" %
%   B12:4/12  "Runout Do Not Use Height Sensor" %

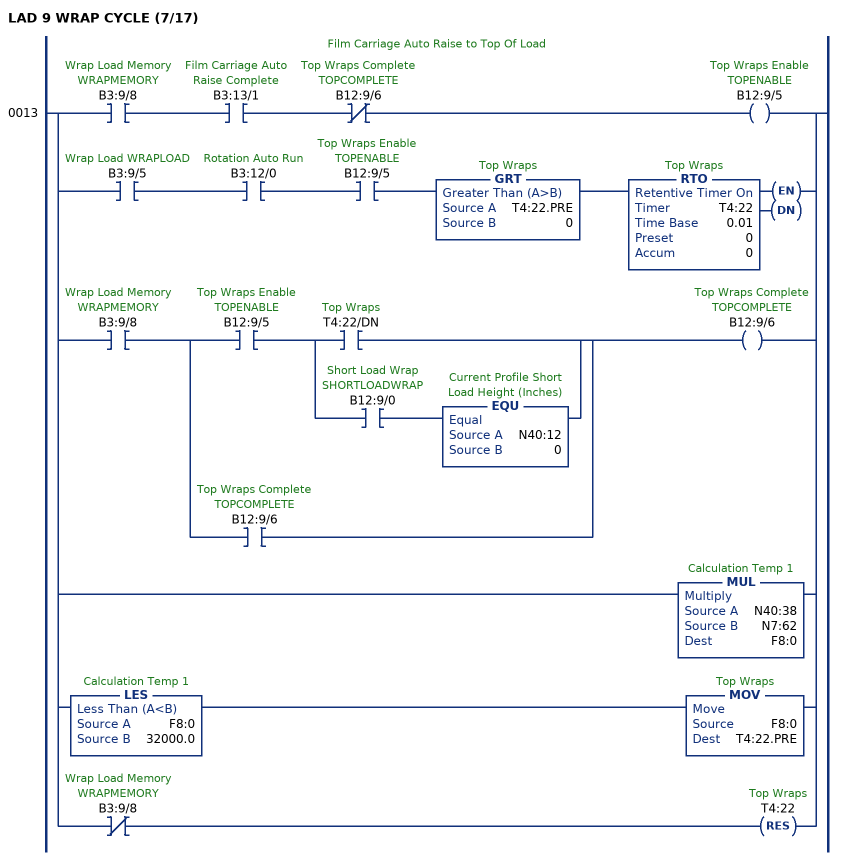
% Rung: 13 %
% Film Carriage Auto Raise to Top Of Load %
SOR BST XIC B3:9/8 XIC B3:13/1 XIO B12:9/6 OTE B12:9/5 NXB XIC B3:9/5 XIC B3:12/0 XIC B12:9/5 GRT T4:22.PRE 0 RTO T4:22 0.01 0 0 NXB XIC B3:9/8 BST XIC B12:9/5 BST XIC T4:22/DN NXB XIC B12:9/0 EQU N40:12 0 BND NXB XIC B12:9/6 BND OTE B12:9/6 NXB BST MUL N40:38 N7:62 F8:0 NXB LES F8:0 32000.0 MOV F8:0 T4:22.PRE BND NXB XIO B3:9/8 RES T4:22 BND EOR
%   B3:9/8  WRAPMEMORY  "Wrap Load Memory" %
%   B3:13/1  "Film Carriage Auto Raise Complete" %
%   B12:9/6  TOPCOMPLETE  "Top Wraps Complete" %
%   B12:9/5  TOPENABLE  "Top Wraps Enable" %
%   B3:9/5  WRAPLOAD  "Wrap Load" %
%   B3:12/0  "Rotation Auto Run" %
%   T4:22  "Top Wraps" %
%   B12:9/0  SHORTLOADWRAP  "Short Load Wrap" %
%   N40:12  "Current Profile Short Load Height (Inches)" %
%   N7:62  "Rotation Revolution Time (100 = 1.00s)" %
%   F8:0  "Calculation Temp 1" %

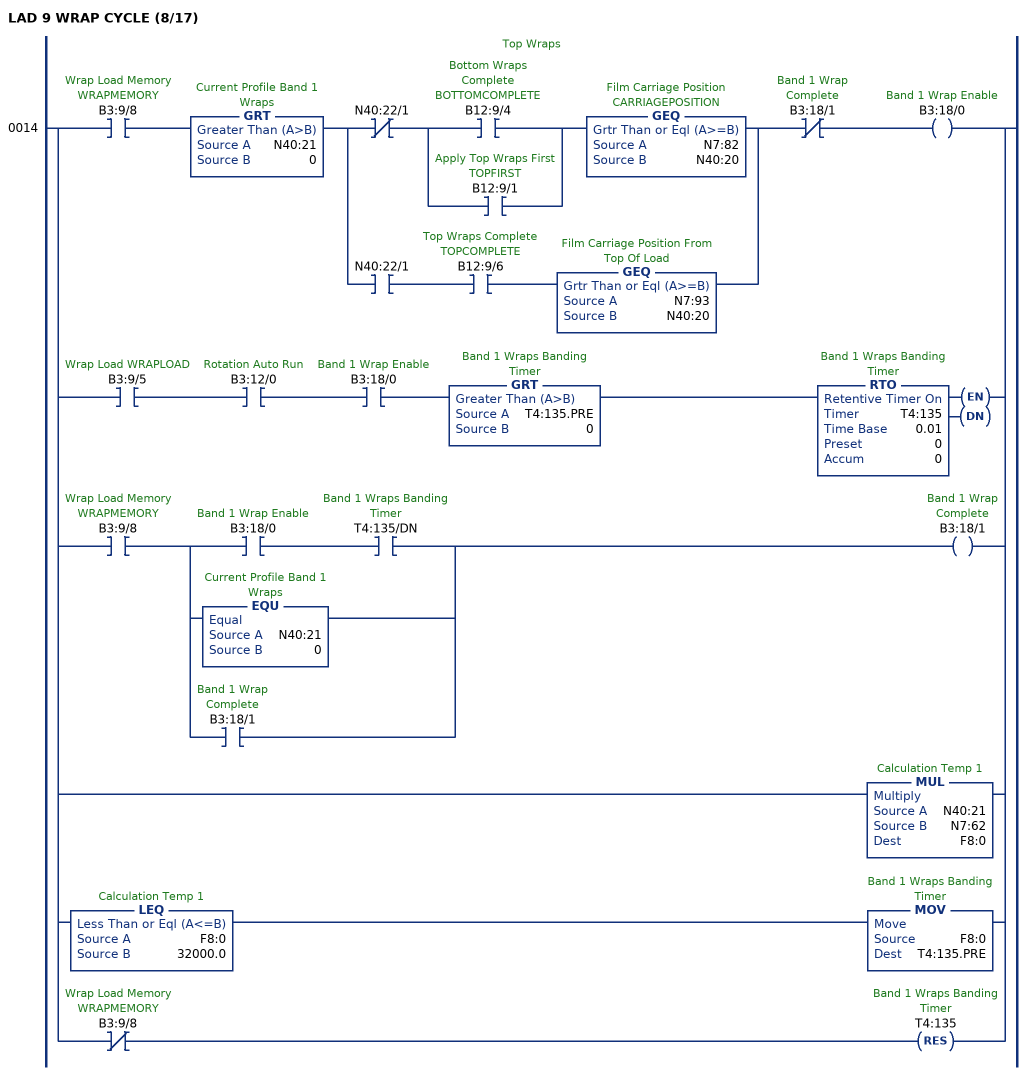
% Rung: 14 %
% Top Wraps %
SOR BST XIC B3:9/8 GRT N40:21 0 BST XIO N40:22/1 BST XIC B12:9/4 NXB XIC B12:9/1 BND GEQ N7:82 N40:20 NXB XIC N40:22/1 XIC B12:9/6 GEQ N7:93 N40:20 BND XIO B3:18/1 OTE B3:18/0 NXB XIC B3:9/5 XIC B3:12/0 XIC B3:18/0 GRT T4:135.PRE 0 RTO T4:135 0.01 0 0 NXB XIC B3:9/8 BST XIC B3:18/0 XIC T4:135/DN NXB EQU N40:21 0 NXB XIC B3:18/1 BND OTE B3:18/1 NXB BST MUL N40:21 N7:62 F8:0 NXB LEQ F8:0 32000.0 MOV F8:0 T4:135.PRE BND NXB XIO B3:9/8 RES T4:135 BND EOR
%   B3:9/8  WRAPMEMORY  "Wrap Load Memory" %
%   N40:21  "Current Profile Band 1 Wraps" %
%   B12:9/4  BOTTOMCOMPLETE  "Bottom Wraps Complete" %
%   B12:9/1  TOPFIRST  "Apply Top Wraps First" %
%   N7:82  CARRIAGEPOSITION  "Film Carriage Position" %
%   N40:20  "Current Profile Band 1 Location" %
%   B12:9/6  TOPCOMPLETE  "Top Wraps Complete" %
%   N7:93  "Film Carriage Position From Top Of Load" %
%   B3:18/1  "Band 1 Wrap Complete" %
%   B3:18/0  "Band 1 Wrap Enable" %
%   B3:9/5  WRAPLOAD  "Wrap Load" %
%   B3:12/0  "Rotation Auto Run" %
%   T4:135  "Band 1 Wraps Banding Timer" %
%   N7:62  "Rotation Revolution Time (100 = 1.00s)" %
%   F8:0  "Calculation Temp 1" %

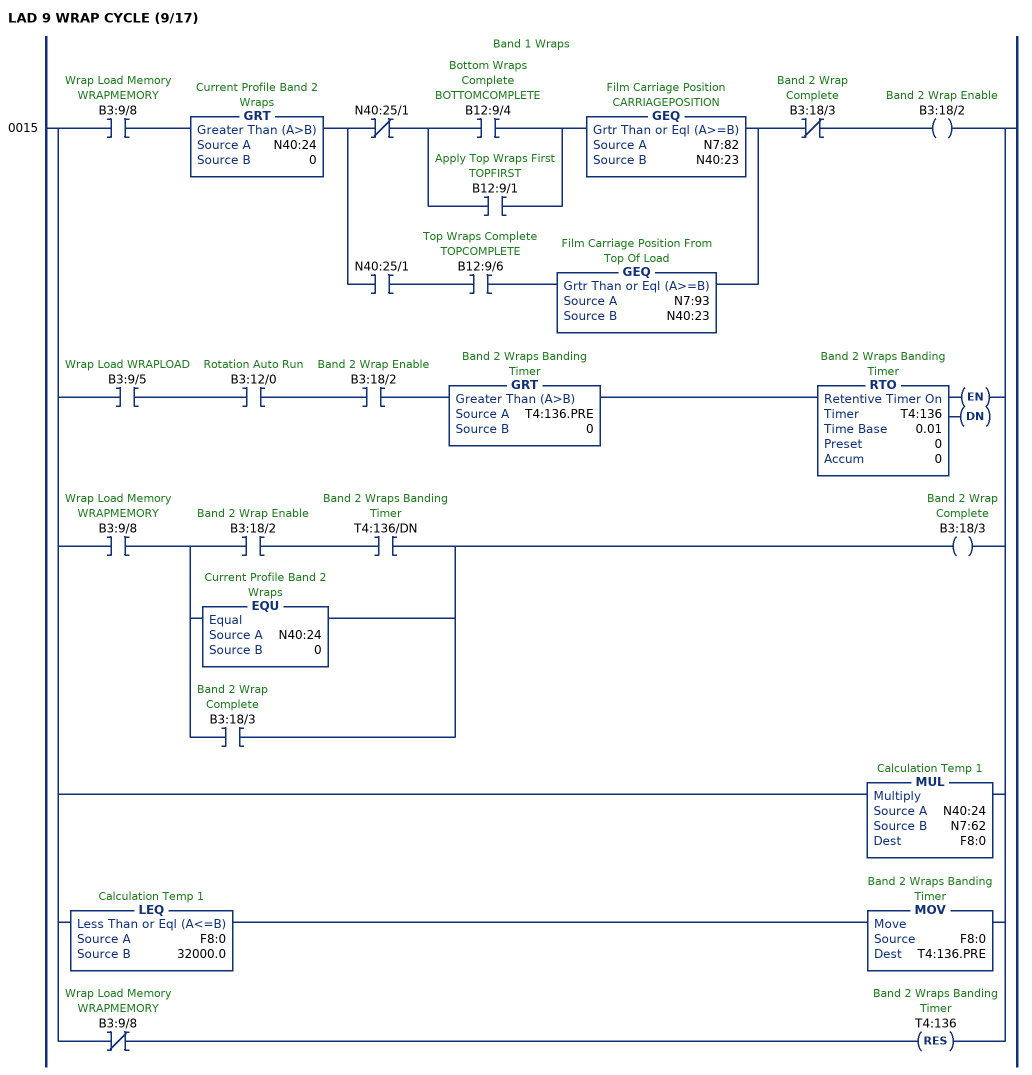
% Rung: 15 %
% Band 1 Wraps %
SOR BST XIC B3:9/8 GRT N40:24 0 BST XIO N40:25/1 BST XIC B12:9/4 NXB XIC B12:9/1 BND GEQ N7:82 N40:23 NXB XIC N40:25/1 XIC B12:9/6 GEQ N7:93 N40:23 BND XIO B3:18/3 OTE B3:18/2 NXB XIC B3:9/5 XIC B3:12/0 XIC B3:18/2 GRT T4:136.PRE 0 RTO T4:136 0.01 0 0 NXB XIC B3:9/8 BST XIC B3:18/2 XIC T4:136/DN NXB EQU N40:24 0 NXB XIC B3:18/3 BND OTE B3:18/3 NXB BST MUL N40:24 N7:62 F8:0 NXB LEQ F8:0 32000.0 MOV F8:0 T4:136.PRE BND NXB XIO B3:9/8 RES T4:136 BND EOR
%   B3:9/8  WRAPMEMORY  "Wrap Load Memory" %
%   N40:24  "Current Profile Band 2 Wraps" %
%   B12:9/4  BOTTOMCOMPLETE  "Bottom Wraps Complete" %
%   B12:9/1  TOPFIRST  "Apply Top Wraps First" %
%   N7:82  CARRIAGEPOSITION  "Film Carriage Position" %
%   N40:23  "Current Profile Band 2 Location" %
%   B12:9/6  TOPCOMPLETE  "Top Wraps Complete" %
%   N7:93  "Film Carriage Position From Top Of Load" %
%   B3:18/3  "Band 2 Wrap Complete" %
%   B3:18/2  "Band 2 Wrap Enable" %
%   B3:9/5  WRAPLOAD  "Wrap Load" %
%   B3:12/0  "Rotation Auto Run" %
%   T4:136  "Band 2 Wraps Banding Timer" %
%   N7:62  "Rotation Revolution Time (100 = 1.00s)" %
%   F8:0  "Calculation Temp 1" %

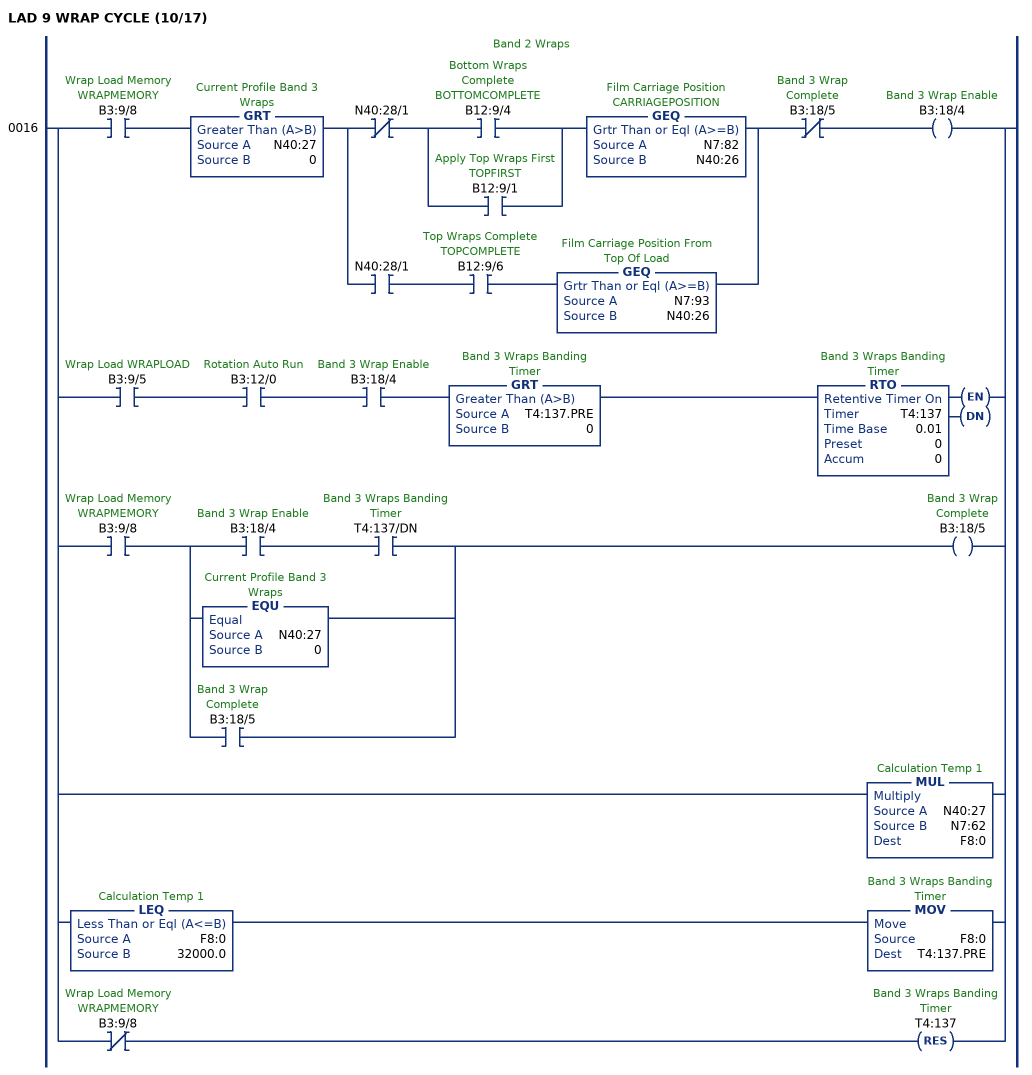
% Rung: 16 %
% Band 2 Wraps %
SOR BST XIC B3:9/8 GRT N40:27 0 BST XIO N40:28/1 BST XIC B12:9/4 NXB XIC B12:9/1 BND GEQ N7:82 N40:26 NXB XIC N40:28/1 XIC B12:9/6 GEQ N7:93 N40:26 BND XIO B3:18/5 OTE B3:18/4 NXB XIC B3:9/5 XIC B3:12/0 XIC B3:18/4 GRT T4:137.PRE 0 RTO T4:137 0.01 0 0 NXB XIC B3:9/8 BST XIC B3:18/4 XIC T4:137/DN NXB EQU N40:27 0 NXB XIC B3:18/5 BND OTE B3:18/5 NXB BST MUL N40:27 N7:62 F8:0 NXB LEQ F8:0 32000.0 MOV F8:0 T4:137.PRE BND NXB XIO B3:9/8 RES T4:137 BND EOR
%   B3:9/8  WRAPMEMORY  "Wrap Load Memory" %
%   N40:27  "Current Profile Band 3 Wraps" %
%   B12:9/4  BOTTOMCOMPLETE  "Bottom Wraps Complete" %
%   B12:9/1  TOPFIRST  "Apply Top Wraps First" %
%   N7:82  CARRIAGEPOSITION  "Film Carriage Position" %
%   N40:26  "Current Profile Band 3 Location" %
%   B12:9/6  TOPCOMPLETE  "Top Wraps Complete" %
%   N7:93  "Film Carriage Position From Top Of Load" %
%   B3:18/5  "Band 3 Wrap Complete" %
%   B3:18/4  "Band 3 Wrap Enable" %
%   B3:9/5  WRAPLOAD  "Wrap Load" %
%   B3:12/0  "Rotation Auto Run" %
%   T4:137  "Band 3 Wraps Banding Timer" %
%   N7:62  "Rotation Revolution Time (100 = 1.00s)" %
%   F8:0  "Calculation Temp 1" %

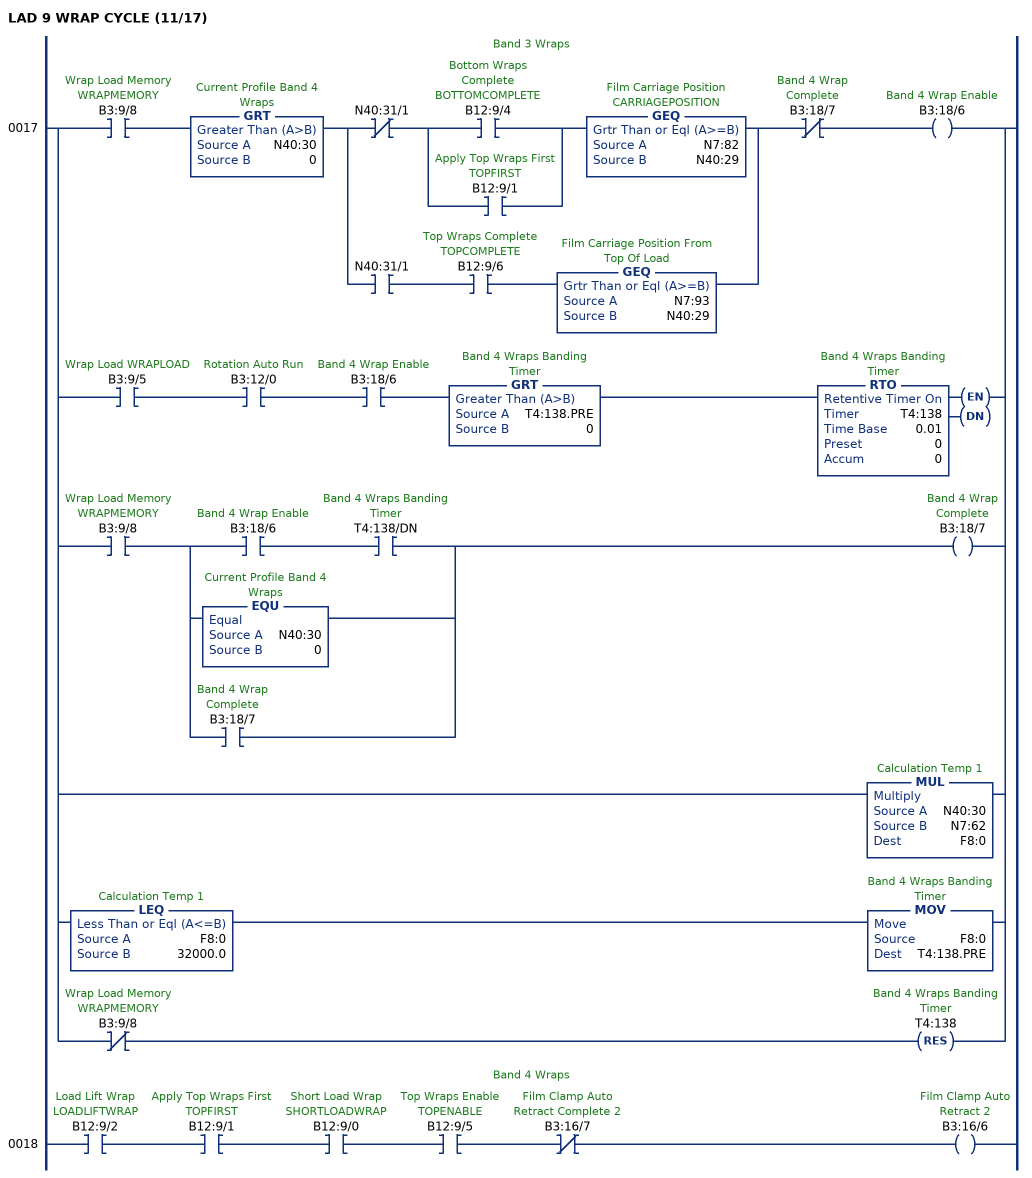
% Rung: 17 %
% Band 3 Wraps %
SOR BST XIC B3:9/8 GRT N40:30 0 BST XIO N40:31/1 BST XIC B12:9/4 NXB XIC B12:9/1 BND GEQ N7:82 N40:29 NXB XIC N40:31/1 XIC B12:9/6 GEQ N7:93 N40:29 BND XIO B3:18/7 OTE B3:18/6 NXB XIC B3:9/5 XIC B3:12/0 XIC B3:18/6 GRT T4:138.PRE 0 RTO T4:138 0.01 0 0 NXB XIC B3:9/8 BST XIC B3:18/6 XIC T4:138/DN NXB EQU N40:30 0 NXB XIC B3:18/7 BND OTE B3:18/7 NXB BST MUL N40:30 N7:62 F8:0 NXB LEQ F8:0 32000.0 MOV F8:0 T4:138.PRE BND NXB XIO B3:9/8 RES T4:138 BND EOR
%   B3:9/8  WRAPMEMORY  "Wrap Load Memory" %
%   N40:30  "Current Profile Band 4 Wraps" %
%   B12:9/4  BOTTOMCOMPLETE  "Bottom Wraps Complete" %
%   B12:9/1  TOPFIRST  "Apply Top Wraps First" %
%   N7:82  CARRIAGEPOSITION  "Film Carriage Position" %
%   N40:29  "Current Profile Band 4 Location" %
%   B12:9/6  TOPCOMPLETE  "Top Wraps Complete" %
%   N7:93  "Film Carriage Position From Top Of Load" %
%   B3:18/7  "Band 4 Wrap Complete" %
%   B3:18/6  "Band 4 Wrap Enable" %
%   B3:9/5  WRAPLOAD  "Wrap Load" %
%   B3:12/0  "Rotation Auto Run" %
%   T4:138  "Band 4 Wraps Banding Timer" %
%   N7:62  "Rotation Revolution Time (100 = 1.00s)" %
%   F8:0  "Calculation Temp 1" %
% Rung: 18 %
% Band 4 Wraps %
SOR XIC B12:9/2 XIC B12:9/1 XIC B12:9/0 XIC B12:9/5 XIO B3:16/7 OTE B3:16/6 EOR
%   B12:9/2  LOADLIFTWRAP  "Load Lift Wrap" %
%   B12:9/1  TOPFIRST  "Apply Top Wraps First" %
%   B12:9/0  SHORTLOADWRAP  "Short Load Wrap" %
%   B12:9/5  TOPENABLE  "Top Wraps Enable" %
%   B3:16/7  "Film Clamp Auto Retract Complete 2" %
%   B3:16/6  "Film Clamp Auto Retract 2" %

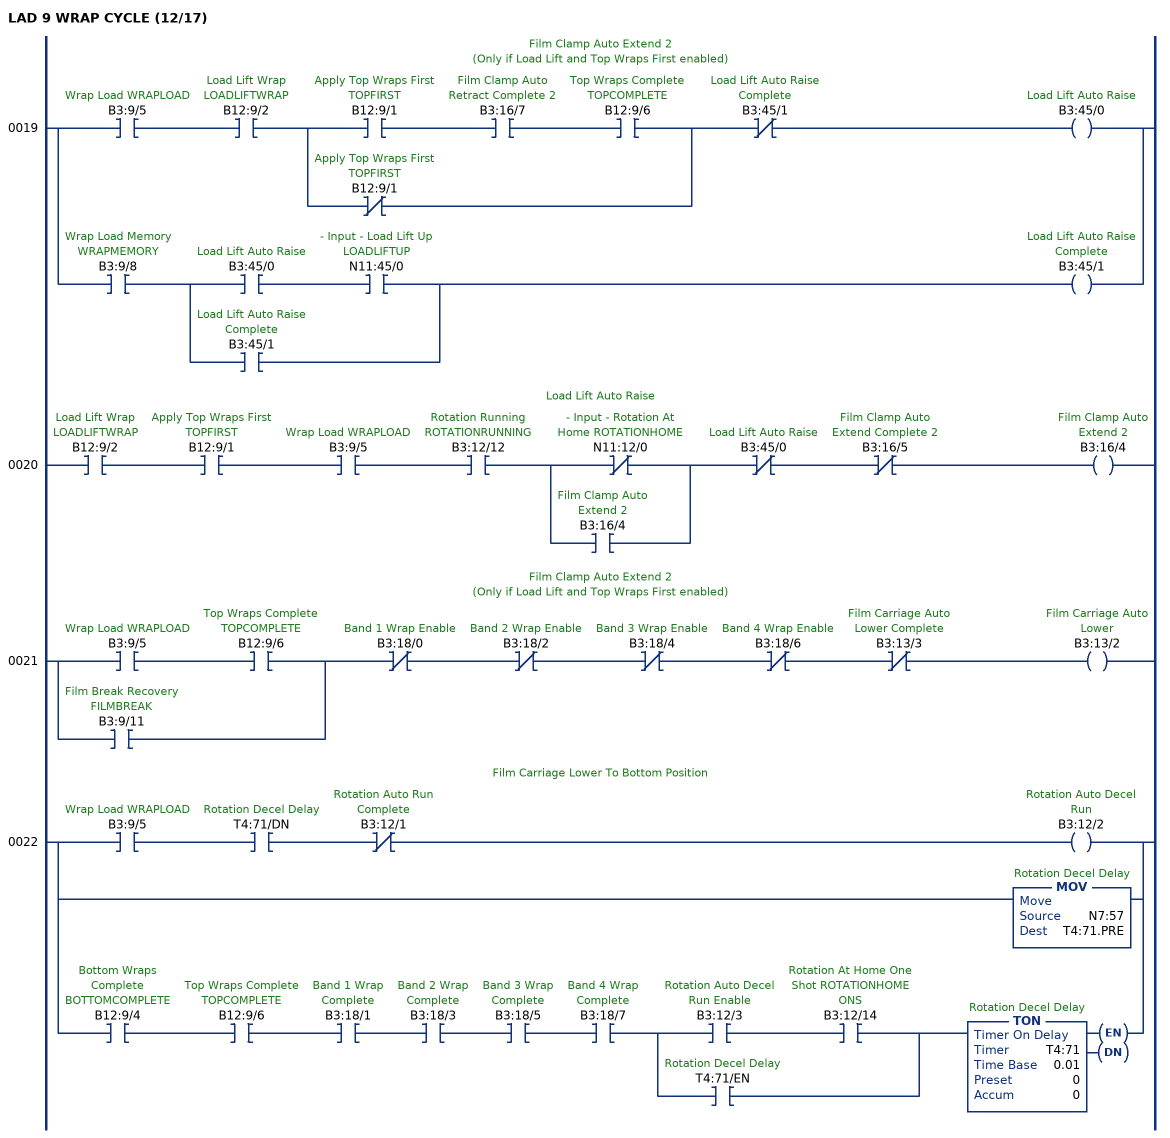
% Rung: 19 %
% Film Clamp Auto Extend 2
% (Only if Load Lift and Top Wraps First enabled) %
SOR BST XIC B3:9/5 XIC B12:9/2 BST XIC B12:9/1 XIC B3:16/7 XIC B12:9/6 NXB XIO B12:9/1 BND XIO B3:45/1 OTE B3:45/0 NXB XIC B3:9/8 BST XIC B3:45/0 XIC N11:45/0 NXB XIC B3:45/1 BND OTE B3:45/1 BND EOR
%   B3:9/5  WRAPLOAD  "Wrap Load" %
%   B12:9/2  LOADLIFTWRAP  "Load Lift Wrap" %
%   B12:9/1  TOPFIRST  "Apply Top Wraps First" %
%   B3:16/7  "Film Clamp Auto Retract Complete 2" %
%   B12:9/6  TOPCOMPLETE  "Top Wraps Complete" %
%   B3:45/1  "Load Lift Auto Raise Complete" %
%   B3:45/0  "Load Lift Auto Raise" %
%   B3:9/8  WRAPMEMORY  "Wrap Load Memory" %
%   N11:45/0  LOADLIFTUP  "- Input - Load Lift Up" %
% Rung: 20 %
% Load Lift Auto Raise %
SOR XIC B12:9/2 XIC B12:9/1 XIC B3:9/5 XIC B3:12/12 BST XIO N11:12/0 NXB XIC B3:16/4 BND XIO B3:45/0 XIO B3:16/5 OTE B3:16/4 EOR
%   B12:9/2  LOADLIFTWRAP  "Load Lift Wrap" %
%   B12:9/1  TOPFIRST  "Apply Top Wraps First" %
%   B3:9/5  WRAPLOAD  "Wrap Load" %
%   B3:12/12  ROTATIONRUNNING  "Rotation Running" %
%   N11:12/0  ROTATIONHOME  "- Input - Rotation At Home" %
%   B3:16/4  "Film Clamp Auto Extend 2" %
%   B3:45/0  "Load Lift Auto Raise" %
%   B3:16/5  "Film Clamp Auto Extend Complete 2" %
% Rung: 21 %
% Film Clamp Auto Extend 2
% (Only if Load Lift and Top Wraps First enabled) %
SOR BST XIC B3:9/5 XIC B12:9/6 NXB XIC B3:9/11 BND XIO B3:18/0 XIO B3:18/2 XIO B3:18/4 XIO B3:18/6 XIO B3:13/3 OTE B3:13/2 EOR
%   B3:9/5  WRAPLOAD  "Wrap Load" %
%   B12:9/6  TOPCOMPLETE  "Top Wraps Complete" %
%   B3:9/11  FILMBREAK  "Film Break Recovery" %
%   B3:18/0  "Band 1 Wrap Enable" %
%   B3:18/2  "Band 2 Wrap Enable" %
%   B3:18/4  "Band 3 Wrap Enable" %
%   B3:18/6  "Band 4 Wrap Enable" %
%   B3:13/3  "Film Carriage Auto Lower Complete" %
%   B3:13/2  "Film Carriage Auto Lower" %
% Rung: 22 %
% Film Carriage Lower To Bottom Position %
SOR BST XIC B3:9/5 XIC T4:71/DN XIO B3:12/1 OTE B3:12/2 NXB MOV N7:57 T4:71.PRE NXB XIC B12:9/4 XIC B12:9/6 XIC B3:18/1 XIC B3:18/3 XIC B3:18/5 XIC B3:18/7 BST XIC B3:12/3 XIC B3:12/14 NXB XIC T4:71/EN BND TON T4:71 0.01 0 0 BND EOR
%   B3:9/5  WRAPLOAD  "Wrap Load" %
%   T4:71  "Rotation Decel Delay" %
%   B3:12/1  "Rotation Auto Run Complete" %
%   B3:12/2  "Rotation Auto Decel Run" %
%   N7:57  "Rotation Decel Delay Time (100 = 1.00s)" %
%   B12:9/4  BOTTOMCOMPLETE  "Bottom Wraps Complete" %
%   B12:9/6  TOPCOMPLETE  "Top Wraps Complete" %
%   B3:18/1  "Band 1 Wrap Complete" %
%   B3:18/3  "Band 2 Wrap Complete" %
%   B3:18/5  "Band 3 Wrap Complete" %
%   B3:18/7  "Band 4 Wrap Complete" %
%   B3:12/3  "Rotation Auto Decel Run Enable" %
%   B3:12/14  ROTATIONHOMEONS  "Rotation At Home One Shot" %

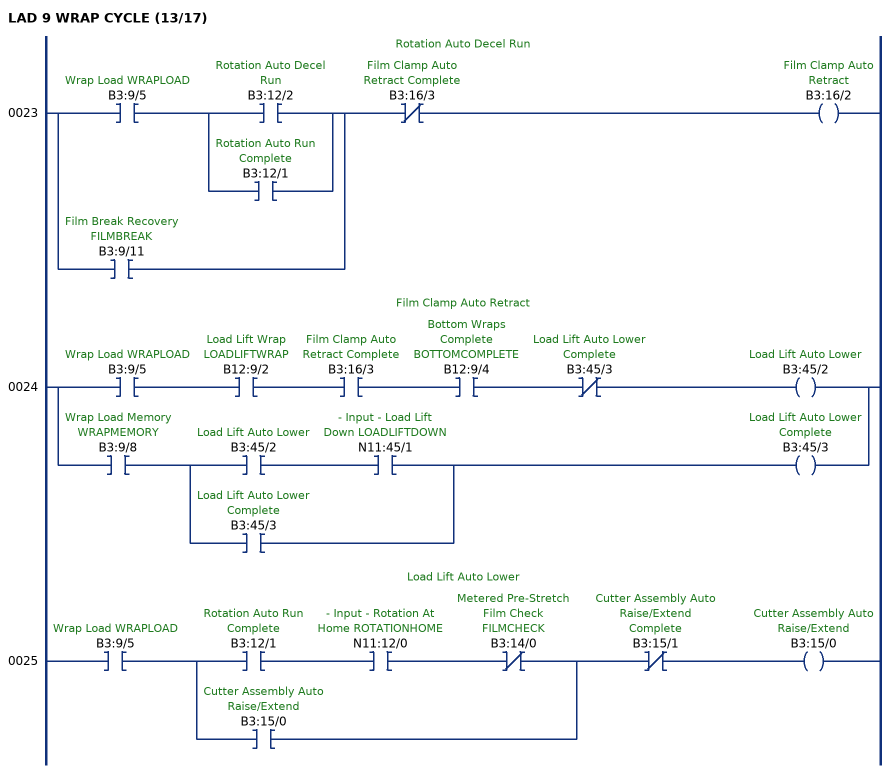
% Rung: 23 %
% Rotation Auto Decel Run %
SOR BST XIC B3:9/5 BST XIC B3:12/2 NXB XIC B3:12/1 BND NXB XIC B3:9/11 BND XIO B3:16/3 OTE B3:16/2 EOR
%   B3:9/5  WRAPLOAD  "Wrap Load" %
%   B3:12/2  "Rotation Auto Decel Run" %
%   B3:12/1  "Rotation Auto Run Complete" %
%   B3:9/11  FILMBREAK  "Film Break Recovery" %
%   B3:16/3  "Film Clamp Auto Retract Complete" %
%   B3:16/2  "Film Clamp Auto Retract" %
% Rung: 24 %
% Film Clamp Auto Retract %
SOR BST XIC B3:9/5 XIC B12:9/2 XIC B3:16/3 XIC B12:9/4 XIO B3:45/3 OTE B3:45/2 NXB XIC B3:9/8 BST XIC B3:45/2 XIC N11:45/1 NXB XIC B3:45/3 BND OTE B3:45/3 BND EOR
%   B3:9/5  WRAPLOAD  "Wrap Load" %
%   B12:9/2  LOADLIFTWRAP  "Load Lift Wrap" %
%   B3:16/3  "Film Clamp Auto Retract Complete" %
%   B12:9/4  BOTTOMCOMPLETE  "Bottom Wraps Complete" %
%   B3:45/3  "Load Lift Auto Lower Complete" %
%   B3:45/2  "Load Lift Auto Lower" %
%   B3:9/8  WRAPMEMORY  "Wrap Load Memory" %
%   N11:45/1  LOADLIFTDOWN  "- Input - Load Lift Down" %
% Rung: 25 %
% Load Lift Auto Lower %
SOR XIC B3:9/5 BST XIC B3:12/1 XIC N11:12/0 XIO B3:14/0 NXB XIC B3:15/0 BND XIO B3:15/1 OTE B3:15/0 EOR
%   B3:9/5  WRAPLOAD  "Wrap Load" %
%   B3:12/1  "Rotation Auto Run Complete" %
%   N11:12/0  ROTATIONHOME  "- Input - Rotation At Home" %
%   B3:14/0  FILMCHECK  "Metered Pre-Stretch Film Check" %
%   B3:15/0  "Cutter Assembly Auto Raise/Extend" %
%   B3:15/1  "Cutter Assembly Auto Raise/Extend Complete" %

